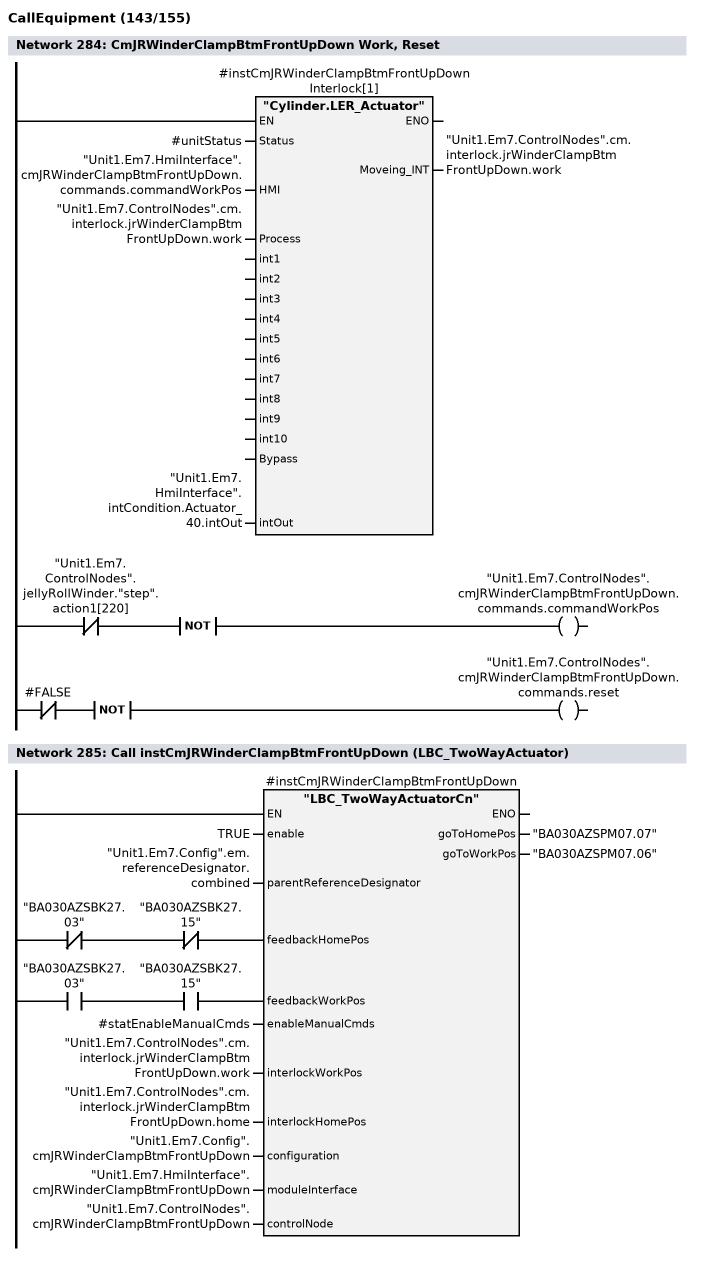
   RUNG wire#powerrail
      #instCmJRWinderClampBtmFrontUpDownInterlock[1](Status := #unitStatus, HMI := "Unit1.Em7.HmiInterface".cmJRWinderClampBtmFrontUpDown.commands.commandWorkPos, Process := "Unit1.Em7.ControlNodes".cm.interlock.jrWinderClampBtmFrontUpDown.work, int1 :=, int2 :=, int3 :=, int4 :=, int5 :=, int6 :=, int7 :=, int8 :=, int9 :=, int10 :=, Bypass :=, intOut := "Unit1.Em7.HmiInterface".intCondition.Actuator_40.intOut, Moveing_INT => "Unit1.Em7.ControlNodes".cm.interlock.jrWinderClampBtmFrontUpDown.work)
   END_RUNG
   RUNG wire#powerrail
      I_Contact( "Unit1.Em7.ControlNodes".jellyRollWinder."step".action1[220] )
      Not()
      Coil( "Unit1.Em7.ControlNodes".cmJRWinderClampBtmFrontUpDown.commands.commandWorkPos )
   END_RUNG
   RUNG wire#powerrail
      I_Contact( #FALSE )
      Not()
      Coil( "Unit1.Em7.ControlNodes".cmJRWinderClampBtmFrontUpDown.commands.reset )
   END_RUNG
   // the same network as SCL:
   #instCmJRWinderClampBtmFrontUpDownInterlock[1](Status := #unitStatus,   // "Cylinder.LER_Actuator"
                           HMI := "Unit1.Em7.HmiInterface".cmJRWinderClampBtmFrontUpDown.commands.commandWorkPos,
                           Process := "Unit1.Em7.ControlNodes".cm.interlock.jrWinderClampBtmFrontUpDown.work,
                           intOut := "Unit1.Em7.HmiInterface".intCondition.Actuator_40.intOut,
                           Moveing_INT => "Unit1.Em7.ControlNodes".cm.interlock.jrWinderClampBtmFrontUpDown.work);
   "Unit1.Em7.ControlNodes".cmJRWinderClampBtmFrontUpDown.commands.commandWorkPos := NOT (NOT "Unit1.Em7.ControlNodes".jellyRollWinder."step".action1[220]);
   "Unit1.Em7.ControlNodes".cmJRWinderClampBtmFrontUpDown.commands.reset := NOT (NOT #FALSE);
END_REGION

REGION Network 285: Call instCmJRWinderClampBtmFrontUpDown (LBC_TwoWayActuator)
   RUNG wire#powerrail
      #instCmJRWinderClampBtmFrontUpDown(feedbackHomePos := wire#w1, feedbackWorkPos := wire#w2, enable := TRUE, parentReferenceDesignator := "Unit1.Em7.Config".em.referenceDesignator.combined, enableManualCmds := #statEnableManualCmds, interlockWorkPos := "Unit1.Em7.ControlNodes".cm.interlock.jrWinderClampBtmFrontUpDown.work, interlockHomePos := "Unit1.Em7.ControlNodes".cm.interlock.jrWinderClampBtmFrontUpDown.home, configuration := "Unit1.Em7.Config".cmJRWinderClampBtmFrontUpDown, moduleInterface := "Unit1.Em7.HmiInterface".cmJRWinderClampBtmFrontUpDown, controlNode := "Unit1.Em7.ControlNodes".cmJRWinderClampBtmFrontUpDown, goToHomePos => "BA030AZSPM07.07", goToWorkPos => "BA030AZSPM07.06")
   END_RUNG
   RUNG wire#powerrail
      I_Contact( "BA030AZSBK27.03" )
      I_Contact( "BA030AZSBK27.15" )
   END_RUNG wire#w1
   RUNG wire#powerrail
      Contact( "BA030AZSBK27.03" )
      Contact( "BA030AZSBK27.15" )
   END_RUNG wire#w2
   // the same network as SCL:
   #instCmJRWinderClampBtmFrontUpDown(enable := TRUE,   // "LBC_TwoWayActuatorCn"
                           parentReferenceDesignator := "Unit1.Em7.Config".em.referenceDesignator.combined,
                           feedbackHomePos := NOT "BA030AZSBK27.03" AND NOT "BA030AZSBK27.15",
                           feedbackWorkPos := "BA030AZSBK27.03" AND "BA030AZSBK27.15",
                           enableManualCmds := #statEnableManualCmds,
                           interlockWorkPos := "Unit1.Em7.ControlNodes".cm.interlock.jrWinderClampBtmFrontUpDown.work,
                           interlockHomePos := "Unit1.Em7.ControlNodes".cm.interlock.jrWinderClampBtmFrontUpDown.home,
                           configuration := "Unit1.Em7.Config".cmJRWinderClampBtmFrontUpDown,
                           moduleInterface := "Unit1.Em7.HmiInterface".cmJRWinderClampBtmFrontUpDown,
                           controlNode := "Unit1.Em7.ControlNodes".cmJRWinderClampBtmFrontUpDown,
                           goToHomePos => "BA030AZSPM07.07",
                           goToWorkPos => "BA030AZSPM07.06");
END_REGION

REGION Network 287: CmPusherRollerFwdBwd Home
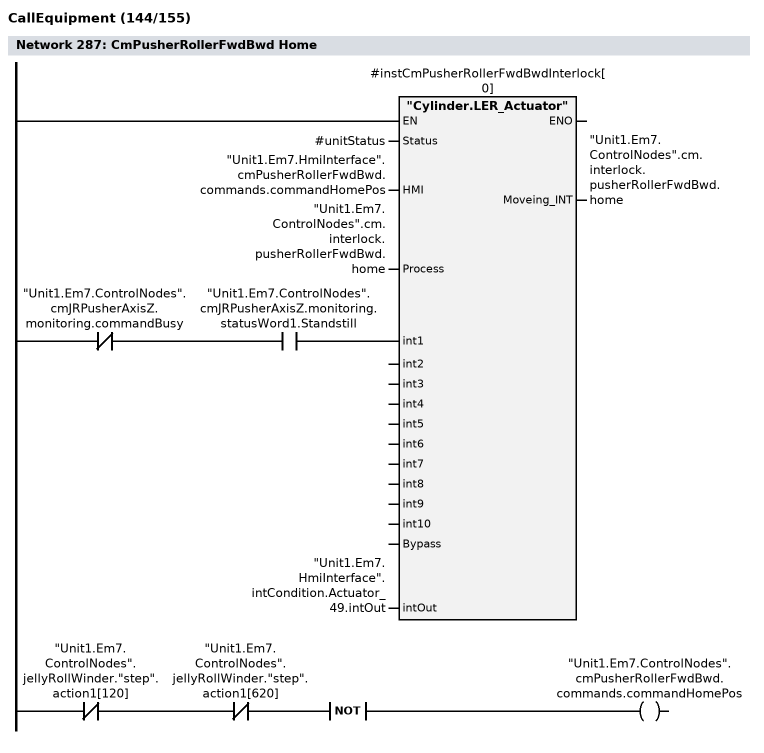
   RUNG wire#powerrail
      #instCmPusherRollerFwdBwdInterlock[0](int1 := wire#w1, Status := #unitStatus, HMI := "Unit1.Em7.HmiInterface".cmPusherRollerFwdBwd.commands.commandHomePos, Process := "Unit1.Em7.ControlNodes".cm.interlock.pusherRollerFwdBwd.home, int2 :=, int3 :=, int4 :=, int5 :=, int6 :=, int7 :=, int8 :=, int9 :=, int10 :=, Bypass :=, intOut := "Unit1.Em7.HmiInterface".intCondition.Actuator_49.intOut, Moveing_INT => "Unit1.Em7.ControlNodes".cm.interlock.pusherRollerFwdBwd.home)
   END_RUNG
   RUNG wire#powerrail
      I_Contact( "Unit1.Em7.ControlNodes".cmJRPusherAxisZ.monitoring.commandBusy )
      Contact( "Unit1.Em7.ControlNodes".cmJRPusherAxisZ.monitoring.statusWord1.Standstill )
   END_RUNG wire#w1
   RUNG wire#powerrail
      I_Contact( "Unit1.Em7.ControlNodes".jellyRollWinder."step".action1[120] )
      I_Contact( "Unit1.Em7.ControlNodes".jellyRollWinder."step".action1[620] )
      Not()
      Coil( "Unit1.Em7.ControlNodes".cmPusherRollerFwdBwd.commands.commandHomePos )
   END_RUNG
   // the same network as SCL:
   #instCmPusherRollerFwdBwdInterlock[0](Status := #unitStatus,   // "Cylinder.LER_Actuator"
                           HMI := "Unit1.Em7.HmiInterface".cmPusherRollerFwdBwd.commands.commandHomePos,
                           Process := "Unit1.Em7.ControlNodes".cm.interlock.pusherRollerFwdBwd.home,
                           int1 := NOT "Unit1.Em7.ControlNodes".cmJRPusherAxisZ.monitoring.commandBusy AND "Unit1.Em7.ControlNodes".cmJRPusherAxisZ.monitoring.statusWord1.Standstill,
                           intOut := "Unit1.Em7.HmiInterface".intCondition.Actuator_49.intOut,
                           Moveing_INT => "Unit1.Em7.ControlNodes".cm.interlock.pusherRollerFwdBwd.home);
   "Unit1.Em7.ControlNodes".cmPusherRollerFwdBwd.commands.commandHomePos := NOT (NOT "Unit1.Em7.ControlNodes".jellyRollWinder."step".action1[120] AND NOT "Unit1.Em7.ControlNodes".jellyRollWinder."step".action1[620]);
END_REGION

REGION Network 288: CmPusherRollerFwdBwd Work
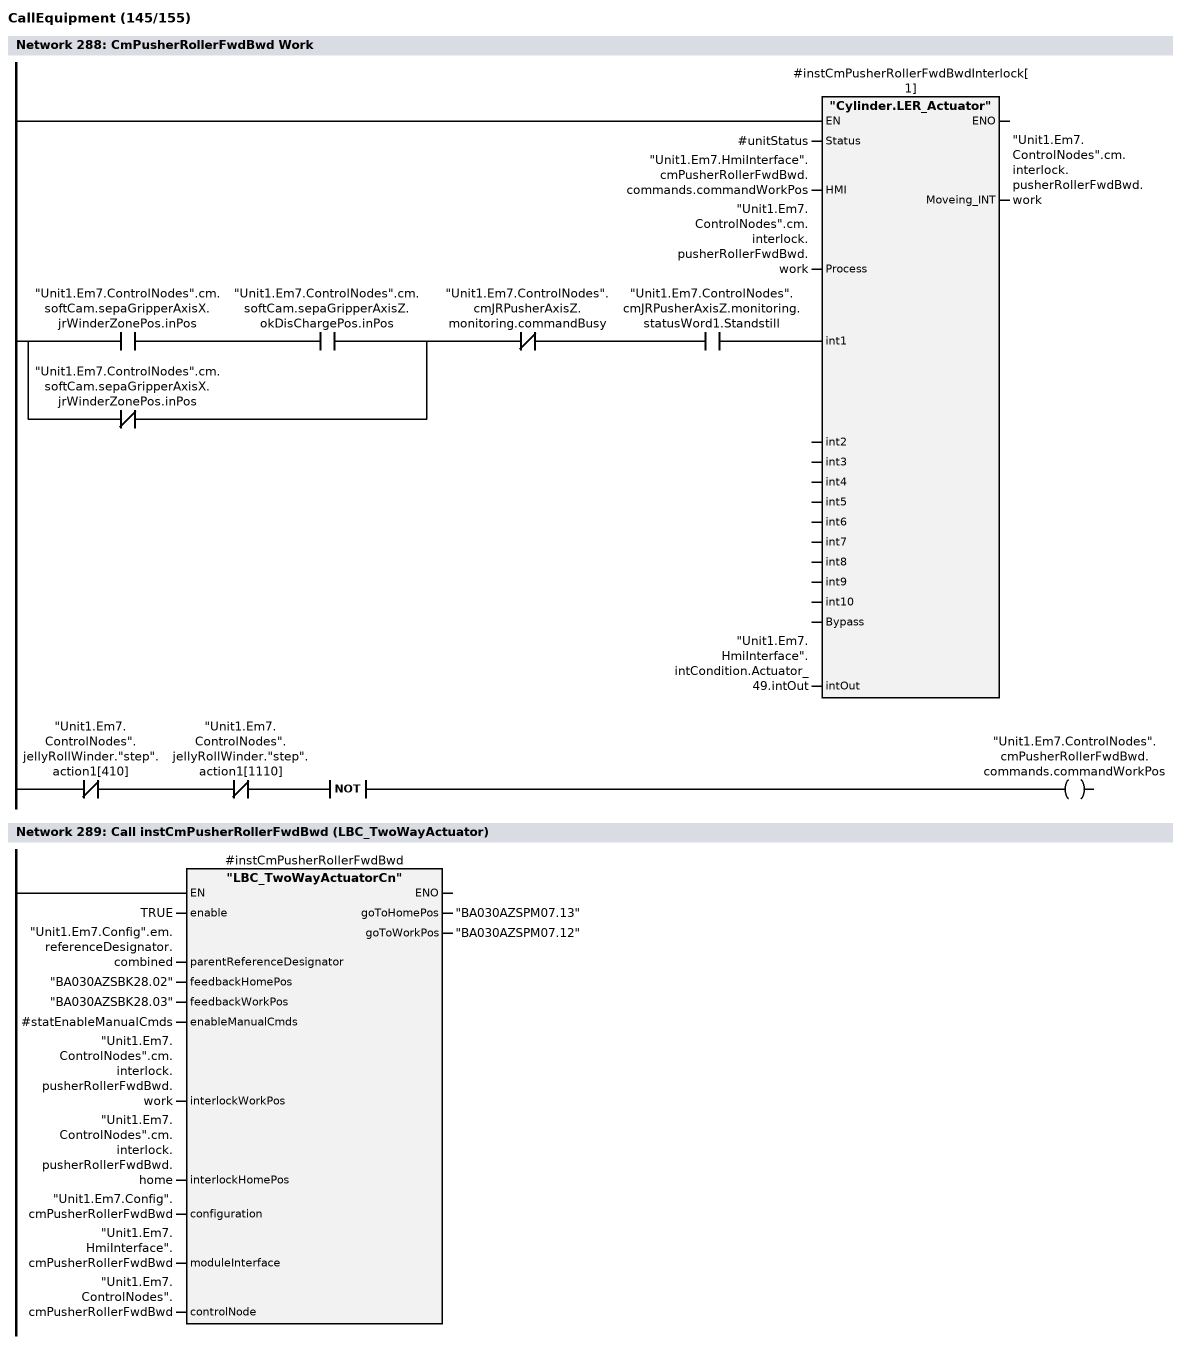
   RUNG wire#powerrail
      #instCmPusherRollerFwdBwdInterlock[1](int1 := wire#w2, Status := #unitStatus, HMI := "Unit1.Em7.HmiInterface".cmPusherRollerFwdBwd.commands.commandWorkPos, Process := "Unit1.Em7.ControlNodes".cm.interlock.pusherRollerFwdBwd.work, int2 :=, int3 :=, int4 :=, int5 :=, int6 :=, int7 :=, int8 :=, int9 :=, int10 :=, Bypass :=, intOut := "Unit1.Em7.HmiInterface".intCondition.Actuator_49.intOut, Moveing_INT => "Unit1.Em7.ControlNodes".cm.interlock.pusherRollerFwdBwd.work)
   END_RUNG
   RUNG wire#powerrail
      Contact( "Unit1.Em7.ControlNodes".cm.softCam.sepaGripperAxisX.jrWinderZonePos.inPos )
      Contact( "Unit1.Em7.ControlNodes".cm.softCam.sepaGripperAxisZ.okDisChargePos.inPos )
      wire#w1
      I_Contact( "Unit1.Em7.ControlNodes".cmJRPusherAxisZ.monitoring.commandBusy )
      Contact( "Unit1.Em7.ControlNodes".cmJRPusherAxisZ.monitoring.statusWord1.Standstill )
   END_RUNG wire#w2
   RUNG wire#powerrail
      I_Contact( "Unit1.Em7.ControlNodes".cm.softCam.sepaGripperAxisX.jrWinderZonePos.inPos )
   END_RUNG wire#w1
   RUNG wire#powerrail
      I_Contact( "Unit1.Em7.ControlNodes".jellyRollWinder."step".action1[410] )
      I_Contact( "Unit1.Em7.ControlNodes".jellyRollWinder."step".action1[1110] )
      Not()
      Coil( "Unit1.Em7.ControlNodes".cmPusherRollerFwdBwd.commands.commandWorkPos )
   END_RUNG
   // the same network as SCL:
   #instCmPusherRollerFwdBwdInterlock[1](Status := #unitStatus,   // "Cylinder.LER_Actuator"
                           HMI := "Unit1.Em7.HmiInterface".cmPusherRollerFwdBwd.commands.commandWorkPos,
                           Process := "Unit1.Em7.ControlNodes".cm.interlock.pusherRollerFwdBwd.work,
                           int1 := (("Unit1.Em7.ControlNodes".cm.softCam.sepaGripperAxisX.jrWinderZonePos.inPos AND "Unit1.Em7.ControlNodes".cm.softCam.sepaGripperAxisZ.okDisChargePos.inPos) OR NOT "Unit1.Em7.ControlNodes".cm.softCam.sepaGripperAxisX.jrWinderZonePos.inPos) AND NOT "Unit1.Em7.ControlNodes".cmJRPusherAxisZ.monitoring.commandBusy AND "Unit1.Em7.ControlNodes".cmJRPusherAxisZ.monitoring.statusWord1.Standstill,
                           intOut := "Unit1.Em7.HmiInterface".intCondition.Actuator_49.intOut,
                           Moveing_INT => "Unit1.Em7.ControlNodes".cm.interlock.pusherRollerFwdBwd.work);
   "Unit1.Em7.ControlNodes".cmPusherRollerFwdBwd.commands.commandWorkPos := NOT (NOT "Unit1.Em7.ControlNodes".jellyRollWinder."step".action1[410] AND NOT "Unit1.Em7.ControlNodes".jellyRollWinder."step".action1[1110]);
END_REGION

REGION Network 289: Call instCmPusherRollerFwdBwd (LBC_TwoWayActuator)
   RUNG wire#powerrail
      #instCmPusherRollerFwdBwd(enable := TRUE, parentReferenceDesignator := "Unit1.Em7.Config".em.referenceDesignator.combined, feedbackHomePos := "BA030AZSBK28.02", feedbackWorkPos := "BA030AZSBK28.03", enableManualCmds := #statEnableManualCmds, interlockWorkPos := "Unit1.Em7.ControlNodes".cm.interlock.pusherRollerFwdBwd.work, interlockHomePos := "Unit1.Em7.ControlNodes".cm.interlock.pusherRollerFwdBwd.home, configuration := "Unit1.Em7.Config".cmPusherRollerFwdBwd, moduleInterface := "Unit1.Em7.HmiInterface".cmPusherRollerFwdBwd, controlNode := "Unit1.Em7.ControlNodes".cmPusherRollerFwdBwd, goToHomePos => "BA030AZSPM07.13", goToWorkPos => "BA030AZSPM07.12")
   END_RUNG
   // the same network as SCL:
   #instCmPusherRollerFwdBwd(enable := TRUE,   // "LBC_TwoWayActuatorCn"
                           parentReferenceDesignator := "Unit1.Em7.Config".em.referenceDesignator.combined,
                           feedbackHomePos := "BA030AZSBK28.02",
                           feedbackWorkPos := "BA030AZSBK28.03",
                           enableManualCmds := #statEnableManualCmds,
                           interlockWorkPos := "Unit1.Em7.ControlNodes".cm.interlock.pusherRollerFwdBwd.work,
                           interlockHomePos := "Unit1.Em7.ControlNodes".cm.interlock.pusherRollerFwdBwd.home,
                           configuration := "Unit1.Em7.Config".cmPusherRollerFwdBwd,
                           moduleInterface := "Unit1.Em7.HmiInterface".cmPusherRollerFwdBwd,
                           controlNode := "Unit1.Em7.ControlNodes".cmPusherRollerFwdBwd,
                           goToHomePos => "BA030AZSPM07.13",
                           goToWorkPos => "BA030AZSPM07.12");
END_REGION

REGION Network 291: ********** Feedback to Unit **********
END_REGION

REGION Network 292: Determine StateComplete (SC) in Mode Production
   // Conditions for the Equipment Modules "stateComplete" feedback to the unit. This feedback is given when the task in for the respective state is complete.
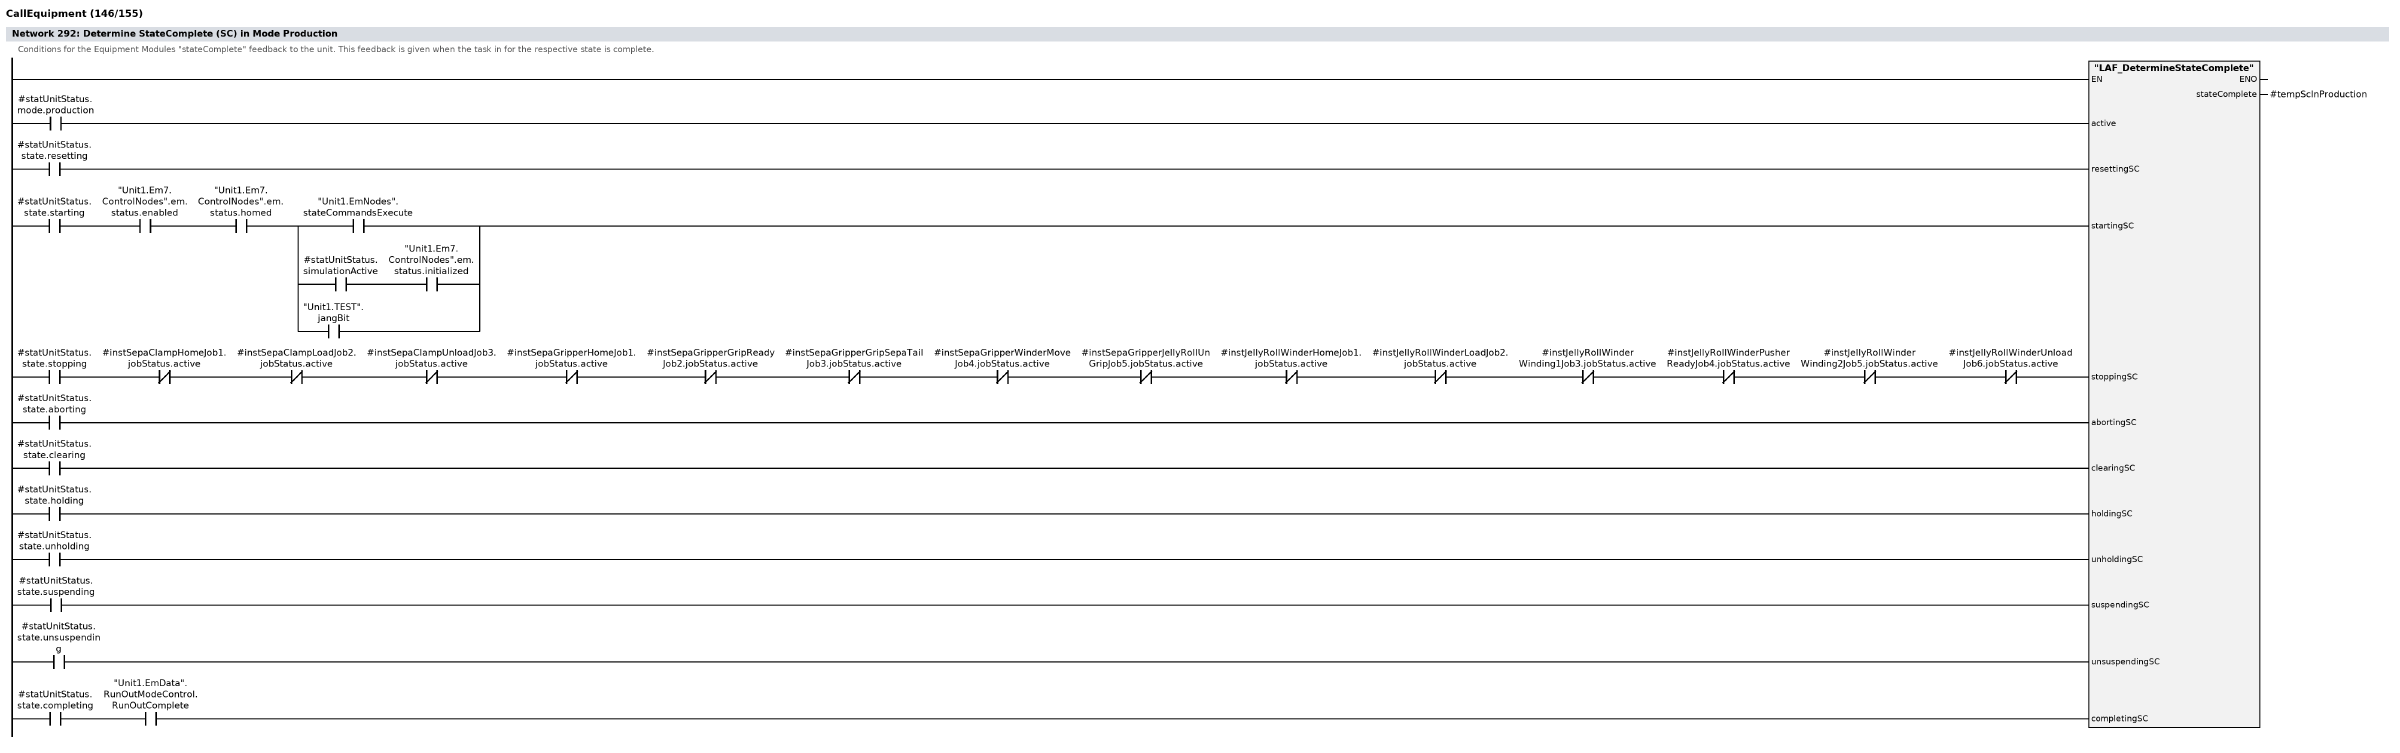
   RUNG wire#powerrail
      "LAF_DetermineStateComplete"(active := wire#w1, resettingSC := wire#w2, startingSC := wire#w4, stoppingSC := wire#w5, abortingSC := wire#w6, clearingSC := wire#w7, holdingSC := wire#w8, unholdingSC := wire#w9, suspendingSC := wire#w10, unsuspendingSC := wire#w11, completingSC := wire#w12, stateComplete => #tempScInProduction)
   END_RUNG
   RUNG wire#powerrail
      Contact( #statUnitStatus.mode.production )
   END_RUNG wire#w1
   RUNG wire#powerrail
      Contact( #statUnitStatus.state.resetting )
   END_RUNG wire#w2
   RUNG wire#powerrail
      Contact( #statUnitStatus.state.starting )
      Contact( "Unit1.Em7.ControlNodes".em.status.enabled )
      Contact( "Unit1.Em7.ControlNodes".em.status.homed )
      wire#w3
      Contact( "Unit1.EmNodes".stateCommandsExecute )
   END_RUNG wire#w4
   RUNG wire#w3
      Contact( #statUnitStatus.simulationActive )
      Contact( "Unit1.Em7.ControlNodes".em.status.initialized )
   END_RUNG wire#w4
   RUNG wire#w3
      Contact( "Unit1.TEST".jangBit )
   END_RUNG wire#w4
   RUNG wire#powerrail
      Contact( #statUnitStatus.state.stopping )
      I_Contact( #instSepaClampHomeJob1.jobStatus.active )
      I_Contact( #instSepaClampLoadJob2.jobStatus.active )
      I_Contact( #instSepaClampUnloadJob3.jobStatus.active )
      I_Contact( #instSepaGripperHomeJob1.jobStatus.active )
      I_Contact( #instSepaGripperGripReadyJob2.jobStatus.active )
      I_Contact( #instSepaGripperGripSepaTailJob3.jobStatus.active )
      I_Contact( #instSepaGripperWinderMoveJob4.jobStatus.active )
      I_Contact( #instSepaGripperJellyRollUnGripJob5.jobStatus.active )
      I_Contact( #instJellyRollWinderHomeJob1.jobStatus.active )
      I_Contact( #instJellyRollWinderLoadJob2.jobStatus.active )
      I_Contact( #instJellyRollWinderWinding1Job3.jobStatus.active )
      I_Contact( #instJellyRollWinderPusherReadyJob4.jobStatus.active )
      I_Contact( #instJellyRollWinderWinding2Job5.jobStatus.active )
      I_Contact( #instJellyRollWinderUnloadJob6.jobStatus.active )
   END_RUNG wire#w5
   RUNG wire#powerrail
      Contact( #statUnitStatus.state.aborting )
   END_RUNG wire#w6
   RUNG wire#powerrail
      Contact( #statUnitStatus.state.clearing )
   END_RUNG wire#w7
   RUNG wire#powerrail
      Contact( #statUnitStatus.state.holding )
   END_RUNG wire#w8
   RUNG wire#powerrail
      Contact( #statUnitStatus.state.unholding )
   END_RUNG wire#w9
   RUNG wire#powerrail
      Contact( #statUnitStatus.state.suspending )
   END_RUNG wire#w10
   RUNG wire#powerrail
      Contact( #statUnitStatus.state.unsuspending )
   END_RUNG wire#w11
   RUNG wire#powerrail
      Contact( #statUnitStatus.state.completing )
      Contact( "Unit1.EmData".RunOutModeControl.RunOutComplete )
   END_RUNG wire#w12
   // the same network as SCL:
   "LAF_DetermineStateComplete"(active := #statUnitStatus.mode.production,
                           resettingSC := #statUnitStatus.state.resetting,
                           startingSC := #statUnitStatus.state.starting AND "Unit1.Em7.ControlNodes".em.status.enabled AND "Unit1.Em7.ControlNodes".em.status.homed AND ("Unit1.EmNodes".stateCommandsExecute OR (#statUnitStatus.simulationActive AND "Unit1.Em7.ControlNodes".em.status.initialized) OR "Unit1.TEST".jangBit),
                           stoppingSC := #statUnitStatus.state.stopping AND NOT #instSepaClampHomeJob1.jobStatus.active AND NOT #instSepaClampLoadJob2.jobStatus.active AND NOT #instSepaClampUnloadJob3.jobStatus.active AND NOT #instSepaGripperHomeJob1.jobStatus.active AND NOT #instSepaGripperGripReadyJob2.jobStatus.active AND NOT #instSepaGripperGripSepaTailJob3.jobStatus.active AND NOT #instSepaGripperWinderMoveJob4.jobStatus.active AND NOT #instSepaGripperJellyRollUnGripJob5.jobStatus.active AND NOT #instJellyRollWinderHomeJob1.jobStatus.active AND NOT #instJellyRollWinderLoadJob2.jobStatus.active AND NOT #instJellyRollWinderWinding1Job3.jobStatus.active AND NOT #instJellyRollWinderPusherReadyJob4.jobStatus.active AND NOT #instJellyRollWinderWinding2Job5.jobStatus.active AND NOT #instJellyRollWinderUnloadJob6.jobStatus.active,
                           abortingSC := #statUnitStatus.state.aborting,
                           clearingSC := #statUnitStatus.state.clearing,
                           holdingSC := #statUnitStatus.state.holding,
                           unholdingSC := #statUnitStatus.state.unholding,
                           suspendingSC := #statUnitStatus.state.suspending,
                           unsuspendingSC := #statUnitStatus.state.unsuspending,
                           completingSC := #statUnitStatus.state.completing AND "Unit1.EmData".RunOutModeControl.RunOutComplete,
                           stateComplete => #tempScInProduction);
END_REGION

REGION Network 293: Determine StateComplete (SC) in Mode Maintenance/Manual
   // Conditions for the Equipment Modules "stateComplete" feedback to the unit. This feedback is given when the task in for the respective state is complete.
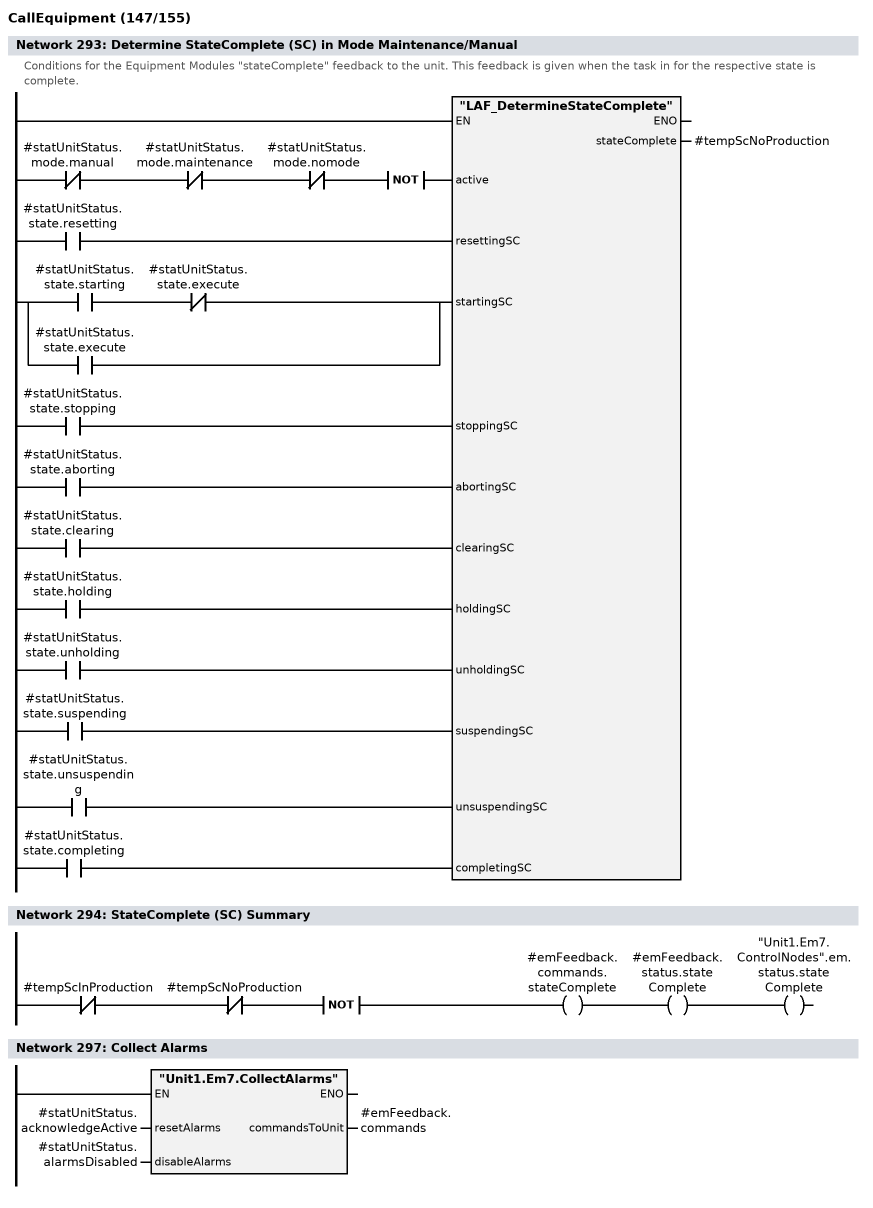
   RUNG wire#powerrail
      "LAF_DetermineStateComplete"(active := wire#w1, resettingSC := wire#w2, startingSC := wire#w3, stoppingSC := wire#w4, abortingSC := wire#w5, clearingSC := wire#w6, holdingSC := wire#w7, unholdingSC := wire#w8, suspendingSC := wire#w9, unsuspendingSC := wire#w10, completingSC := wire#w11, stateComplete => #tempScNoProduction)
   END_RUNG
   RUNG wire#powerrail
      I_Contact( #statUnitStatus.mode.manual )
      I_Contact( #statUnitStatus.mode.maintenance )
      I_Contact( #statUnitStatus.mode.nomode )
      Not()
   END_RUNG wire#w1
   RUNG wire#powerrail
      Contact( #statUnitStatus.state.resetting )
   END_RUNG wire#w2
   RUNG wire#powerrail
      Contact( #statUnitStatus.state.starting )
      I_Contact( #statUnitStatus.state.execute )
   END_RUNG wire#w3
   RUNG wire#powerrail
      Contact( #statUnitStatus.state.execute )
   END_RUNG wire#w3
   RUNG wire#powerrail
      Contact( #statUnitStatus.state.stopping )
   END_RUNG wire#w4
   RUNG wire#powerrail
      Contact( #statUnitStatus.state.aborting )
   END_RUNG wire#w5
   RUNG wire#powerrail
      Contact( #statUnitStatus.state.clearing )
   END_RUNG wire#w6
   RUNG wire#powerrail
      Contact( #statUnitStatus.state.holding )
   END_RUNG wire#w7
   RUNG wire#powerrail
      Contact( #statUnitStatus.state.unholding )
   END_RUNG wire#w8
   RUNG wire#powerrail
      Contact( #statUnitStatus.state.suspending )
   END_RUNG wire#w9
   RUNG wire#powerrail
      Contact( #statUnitStatus.state.unsuspending )
   END_RUNG wire#w10
   RUNG wire#powerrail
      Contact( #statUnitStatus.state.completing )
   END_RUNG wire#w11
   // the same network as SCL:
   "LAF_DetermineStateComplete"(active := NOT (NOT #statUnitStatus.mode.manual AND NOT #statUnitStatus.mode.maintenance AND NOT #statUnitStatus.mode.nomode),
                           resettingSC := #statUnitStatus.state.resetting,
                           startingSC := (#statUnitStatus.state.starting AND NOT #statUnitStatus.state.execute) OR #statUnitStatus.state.execute,
                           stoppingSC := #statUnitStatus.state.stopping,
                           abortingSC := #statUnitStatus.state.aborting,
                           clearingSC := #statUnitStatus.state.clearing,
                           holdingSC := #statUnitStatus.state.holding,
                           unholdingSC := #statUnitStatus.state.unholding,
                           suspendingSC := #statUnitStatus.state.suspending,
                           unsuspendingSC := #statUnitStatus.state.unsuspending,
                           completingSC := #statUnitStatus.state.completing,
                           stateComplete => #tempScNoProduction);
END_REGION

REGION Network 294: StateComplete (SC) Summary
   RUNG wire#powerrail
      I_Contact( #tempScInProduction )
      I_Contact( #tempScNoProduction )
      Not()
      Coil( #emFeedback.commands.stateComplete )
      Coil( #emFeedback.status.stateComplete )
      Coil( "Unit1.Em7.ControlNodes".em.status.stateComplete )
   END_RUNG
   // the same network as SCL:
   #emFeedback.commands.stateComplete := NOT (NOT #tempScInProduction AND NOT #tempScNoProduction);
   #emFeedback.status.stateComplete := #emFeedback.commands.stateComplete;
   "Unit1.Em7.ControlNodes".em.status.stateComplete := #emFeedback.commands.stateComplete;
END_REGION

REGION Network 296: ********** Alarms **********
END_REGION

REGION Network 297: Collect Alarms
   RUNG wire#powerrail
      "Unit1.Em7.CollectAlarms"(resetAlarms := #statUnitStatus.acknowledgeActive, disableAlarms := #statUnitStatus.alarmsDisabled, commandsToUnit => #emFeedback.commands)
   END_RUNG
   // the same network as SCL:
   "Unit1.Em7.CollectAlarms"(resetAlarms := #statUnitStatus.acknowledgeActive,
                           disableAlarms := #statUnitStatus.alarmsDisabled,
                           commandsToUnit => #emFeedback.commands);
END_REGION

REGION Network 298: Manage Alarms
   // Derive commands from the ProDiag supervision. The ProDiag supervisions contain categories which define the reaction of these supervisions (e.g. abort, stop, hold). These are handed over as commands to the unit level.
   // Alternatively, if no ProDiag should be used, you can use the LAF_ManageBitAlarms to realize bit alarm handling. This block can be found in LAF in folder 70_AlarmHandling.
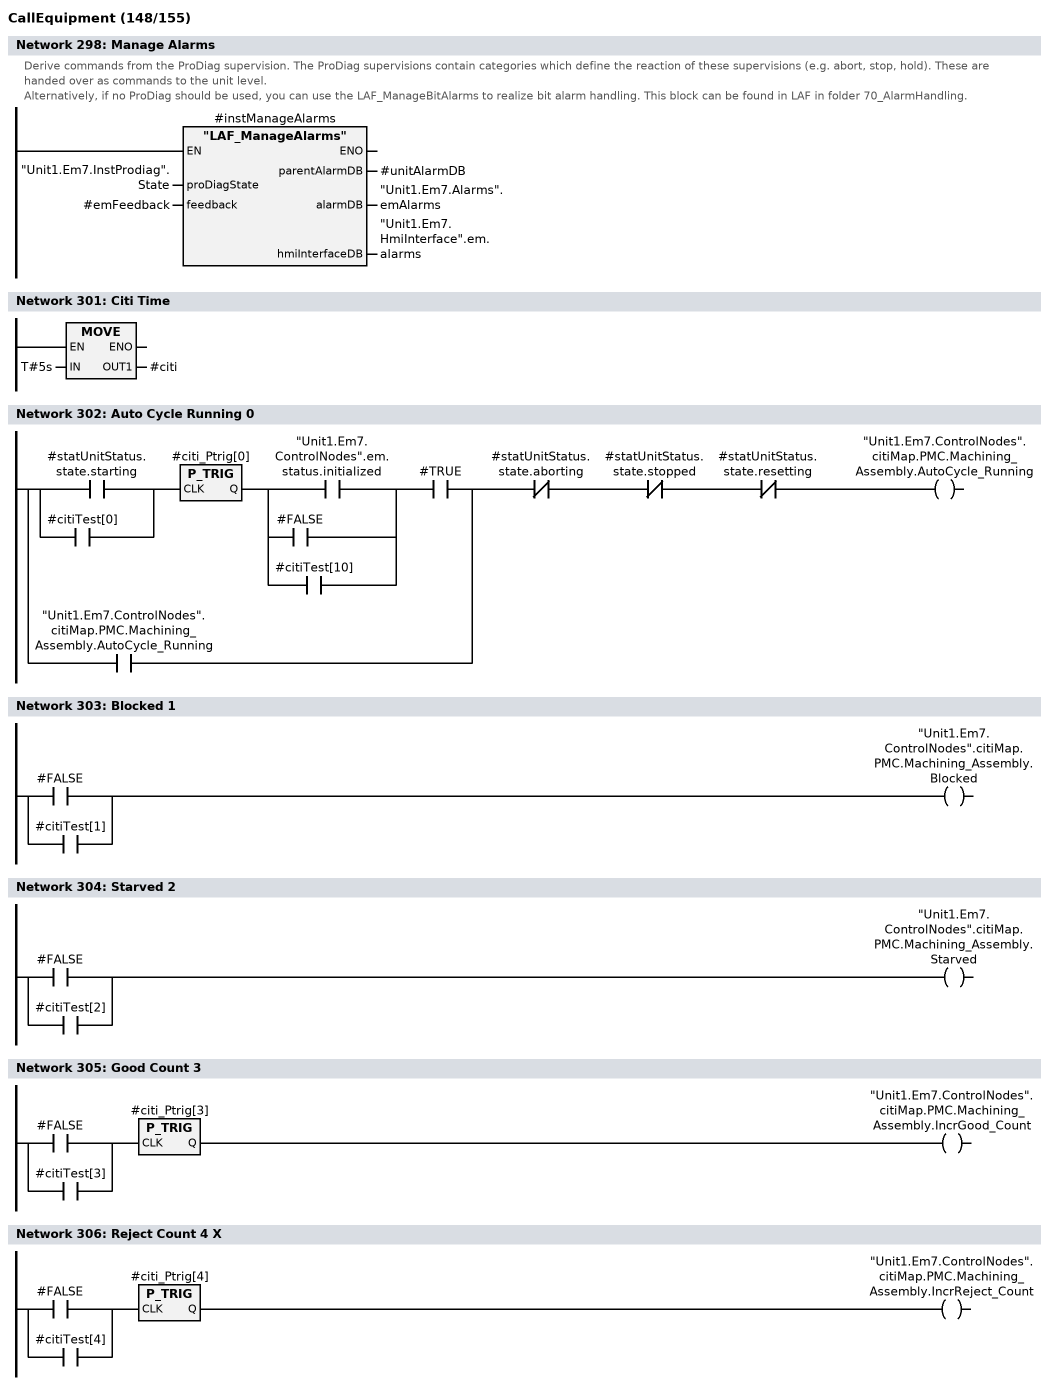
   RUNG wire#powerrail
      #instManageAlarms(proDiagState := "Unit1.Em7.InstProdiag".State, feedback := #emFeedback, parentAlarmDB => #unitAlarmDB, alarmDB => "Unit1.Em7.Alarms".emAlarms, hmiInterfaceDB => "Unit1.Em7.HmiInterface".em.alarms)
   END_RUNG
   // the same network as SCL:
   #instManageAlarms(proDiagState := "Unit1.Em7.InstProdiag".State,   // "LAF_ManageAlarms"
                     feedback := #emFeedback,
                     parentAlarmDB => #unitAlarmDB,
                     alarmDB => "Unit1.Em7.Alarms".emAlarms,
                     hmiInterfaceDB => "Unit1.Em7.HmiInterface".em.alarms);
END_REGION

REGION Network 300: ******************** CITI ********************
END_REGION

REGION Network 301: Citi Time
   RUNG wire#powerrail
      Move(in := T#5s, out1 => #citi)
   END_RUNG
   // the same network as SCL:
   #citi := T#5s;
END_REGION

REGION Network 302: Auto Cycle Running 0
   RUNG wire#powerrail
      Contact( #statUnitStatus.state.starting )
      wire#w1
      P_Trig( #citi_Ptrig[0] )
      wire#w2
      Contact( "Unit1.Em7.ControlNodes".em.status.initialized )
      wire#w3
      Contact( #TRUE )
      wire#w4
      I_Contact( #statUnitStatus.state.aborting )
      I_Contact( #statUnitStatus.state.stopped )
      I_Contact( #statUnitStatus.state.resetting )
      Coil( "Unit1.Em7.ControlNodes".citiMap.PMC.Machining_Assembly.AutoCycle_Running )
   END_RUNG
   RUNG wire#powerrail
      Contact( #citiTest[0] )
   END_RUNG wire#w1
   RUNG wire#w2
      Contact( #FALSE )
   END_RUNG wire#w3
   RUNG wire#w2
      Contact( #citiTest[10] )
   END_RUNG wire#w3
   RUNG wire#powerrail
      Contact( "Unit1.Em7.ControlNodes".citiMap.PMC.Machining_Assembly.AutoCycle_Running )
   END_RUNG wire#w4
   // the same network as SCL:
   #_w1 := #statUnitStatus.state.starting OR #citiTest[0];
   #_w2 := #_w1 AND NOT #citi_Ptrig[0];   // rising edge
   #citi_Ptrig[0] := #_w1;
   "Unit1.Em7.ControlNodes".citiMap.PMC.Machining_Assembly.AutoCycle_Running := ((#_w2 AND ("Unit1.Em7.ControlNodes".em.status.initialized OR #FALSE OR #citiTest[10]) AND #TRUE) OR "Unit1.Em7.ControlNodes".citiMap.PMC.Machining_Assembly.AutoCycle_Running) AND NOT #statUnitStatus.state.aborting AND NOT #statUnitStatus.state.stopped AND NOT #statUnitStatus.state.resetting;
END_REGION

REGION Network 303: Blocked 1
   RUNG wire#powerrail
      Contact( #FALSE )
      wire#w1
      Coil( "Unit1.Em7.ControlNodes".citiMap.PMC.Machining_Assembly.Blocked )
   END_RUNG
   RUNG wire#powerrail
      Contact( #citiTest[1] )
   END_RUNG wire#w1
   // the same network as SCL:
   "Unit1.Em7.ControlNodes".citiMap.PMC.Machining_Assembly.Blocked := #FALSE OR #citiTest[1];
END_REGION

REGION Network 304: Starved 2
   RUNG wire#powerrail
      Contact( #FALSE )
      wire#w1
      Coil( "Unit1.Em7.ControlNodes".citiMap.PMC.Machining_Assembly.Starved )
   END_RUNG
   RUNG wire#powerrail
      Contact( #citiTest[2] )
   END_RUNG wire#w1
   // the same network as SCL:
   "Unit1.Em7.ControlNodes".citiMap.PMC.Machining_Assembly.Starved := #FALSE OR #citiTest[2];
END_REGION

REGION Network 305: Good Count 3
   RUNG wire#powerrail
      Contact( #FALSE )
      wire#w1
      P_Trig( #citi_Ptrig[3] )
      Coil( "Unit1.Em7.ControlNodes".citiMap.PMC.Machining_Assembly.IncrGood_Count )
   END_RUNG
   RUNG wire#powerrail
      Contact( #citiTest[3] )
   END_RUNG wire#w1
   // the same network as SCL:
   #_w1 := #FALSE OR #citiTest[3];
   #_w2 := #_w1 AND NOT #citi_Ptrig[3];   // rising edge
   #citi_Ptrig[3] := #_w1;
   "Unit1.Em7.ControlNodes".citiMap.PMC.Machining_Assembly.IncrGood_Count := #_w2;
END_REGION

REGION Network 306: Reject Count 4 X
   RUNG wire#powerrail
      Contact( #FALSE )
      wire#w1
      P_Trig( #citi_Ptrig[4] )
      Coil( "Unit1.Em7.ControlNodes".citiMap.PMC.Machining_Assembly.IncrReject_Count )
   END_RUNG
   RUNG wire#powerrail
      Contact( #citiTest[4] )
   END_RUNG wire#w1
   // the same network as SCL:
   #_w1 := #FALSE OR #citiTest[4];
   #_w2 := #_w1 AND NOT #citi_Ptrig[4];   // rising edge
   #citi_Ptrig[4] := #_w1;
   "Unit1.Em7.ControlNodes".citiMap.PMC.Machining_Assembly.IncrReject_Count := #_w2;
END_REGION

REGION Network 307: Cycle End Trigger 5
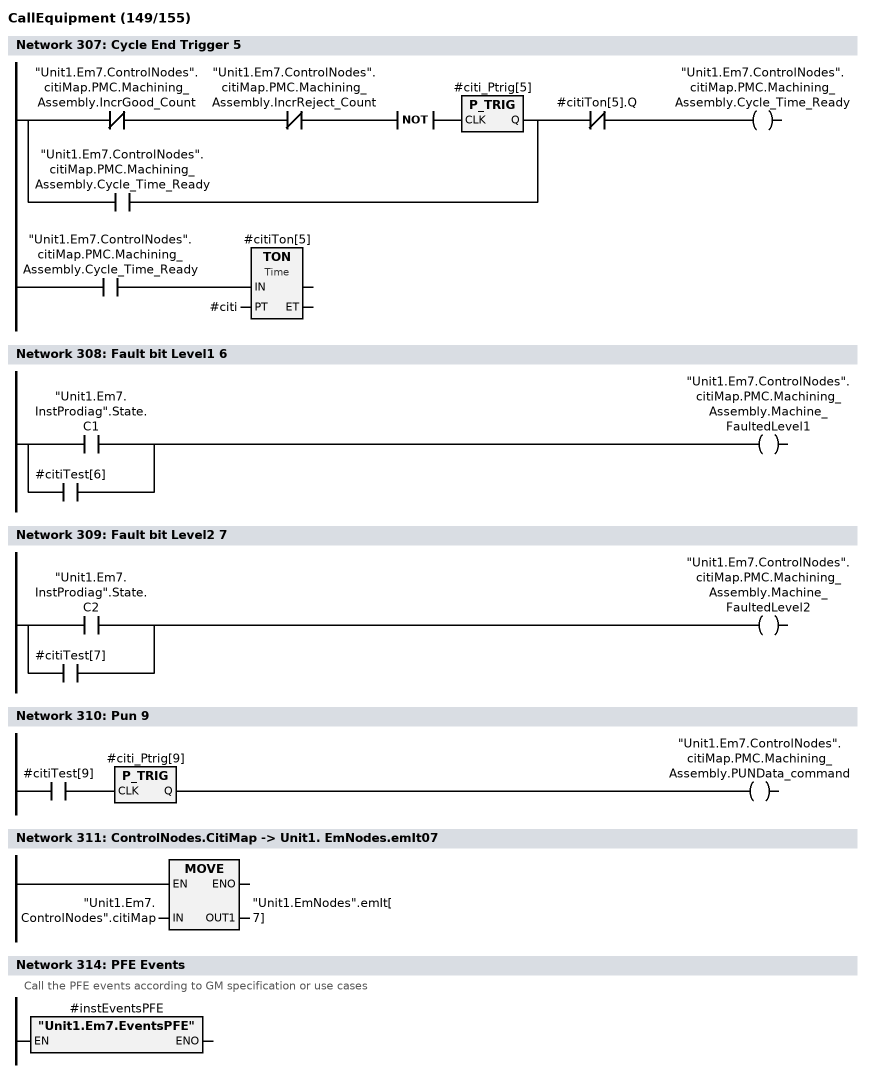
   RUNG wire#powerrail
      I_Contact( "Unit1.Em7.ControlNodes".citiMap.PMC.Machining_Assembly.IncrGood_Count )
      I_Contact( "Unit1.Em7.ControlNodes".citiMap.PMC.Machining_Assembly.IncrReject_Count )
      Not()
      P_Trig( #citi_Ptrig[5] )
      wire#w1
      I_Contact( #citiTon[5].Q )
      Coil( "Unit1.Em7.ControlNodes".citiMap.PMC.Machining_Assembly.Cycle_Time_Ready )
   END_RUNG
   RUNG wire#powerrail
      Contact( "Unit1.Em7.ControlNodes".citiMap.PMC.Machining_Assembly.Cycle_Time_Ready )
   END_RUNG wire#w1
   RUNG wire#powerrail
      Contact( "Unit1.Em7.ControlNodes".citiMap.PMC.Machining_Assembly.Cycle_Time_Ready )
      { S7_Templates := "time_type := Time" } #citiTon[5].TON(pt := #citi, et =>)
   END_RUNG
   // the same network as SCL:
   #_w1 := NOT (NOT "Unit1.Em7.ControlNodes".citiMap.PMC.Machining_Assembly.IncrGood_Count AND NOT "Unit1.Em7.ControlNodes".citiMap.PMC.Machining_Assembly.IncrReject_Count);
   #_w2 := #_w1 AND NOT #citi_Ptrig[5];   // rising edge
   #citi_Ptrig[5] := #_w1;
   "Unit1.Em7.ControlNodes".citiMap.PMC.Machining_Assembly.Cycle_Time_Ready := (#_w2 OR "Unit1.Em7.ControlNodes".citiMap.PMC.Machining_Assembly.Cycle_Time_Ready) AND NOT #citiTon[5].Q;
   #citiTon[5].TON(IN := "Unit1.Em7.ControlNodes".citiMap.PMC.Machining_Assembly.Cycle_Time_Ready, PT := #citi);
END_REGION

REGION Network 308: Fault bit Level1 6
   RUNG wire#powerrail
      Contact( "Unit1.Em7.InstProdiag".State.C1 )
      wire#w1
      Coil( "Unit1.Em7.ControlNodes".citiMap.PMC.Machining_Assembly.Machine_FaultedLevel1 )
   END_RUNG
   RUNG wire#powerrail
      Contact( #citiTest[6] )
   END_RUNG wire#w1
   // the same network as SCL:
   "Unit1.Em7.ControlNodes".citiMap.PMC.Machining_Assembly.Machine_FaultedLevel1 := "Unit1.Em7.InstProdiag".State.C1 OR #citiTest[6];
END_REGION

REGION Network 309: Fault bit Level2 7
   RUNG wire#powerrail
      Contact( "Unit1.Em7.InstProdiag".State.C2 )
      wire#w1
      Coil( "Unit1.Em7.ControlNodes".citiMap.PMC.Machining_Assembly.Machine_FaultedLevel2 )
   END_RUNG
   RUNG wire#powerrail
      Contact( #citiTest[7] )
   END_RUNG wire#w1
   // the same network as SCL:
   "Unit1.Em7.ControlNodes".citiMap.PMC.Machining_Assembly.Machine_FaultedLevel2 := "Unit1.Em7.InstProdiag".State.C2 OR #citiTest[7];
END_REGION

REGION Network 310: Pun 9
   RUNG wire#powerrail
      Contact( #citiTest[9] )
      P_Trig( #citi_Ptrig[9] )
      Coil( "Unit1.Em7.ControlNodes".citiMap.PMC.Machining_Assembly.PUNData_command )
   END_RUNG
   // the same network as SCL:
   #_w1 := #citiTest[9] AND NOT #citi_Ptrig[9];   // rising edge
   #citi_Ptrig[9] := #citiTest[9];
   "Unit1.Em7.ControlNodes".citiMap.PMC.Machining_Assembly.PUNData_command := #_w1;
END_REGION

REGION Network 311: ControlNodes.CitiMap -> Unit1. EmNodes.emIt07
   RUNG wire#powerrail
      Move(in := "Unit1.Em7.ControlNodes".citiMap, out1 => "Unit1.EmNodes".emIt[7])
   END_RUNG
   // the same network as SCL:
   "Unit1.EmNodes".emIt[7] := "Unit1.Em7.ControlNodes".citiMap;
END_REGION

REGION Network 313: ********** PFE Events **********
END_REGION

REGION Network 314: PFE Events
   // Call the PFE events according to GM specification or use cases
   RUNG wire#powerrail
      #instEventsPFE()
   END_RUNG
   // the same network as SCL:
   #instEventsPFE();   // "Unit1.Em7.EventsPFE"
END_REGION

REGION Network 316: ******************** Unit Output ********************
END_REGION

REGION Network 317: Em7 Relations Softcam
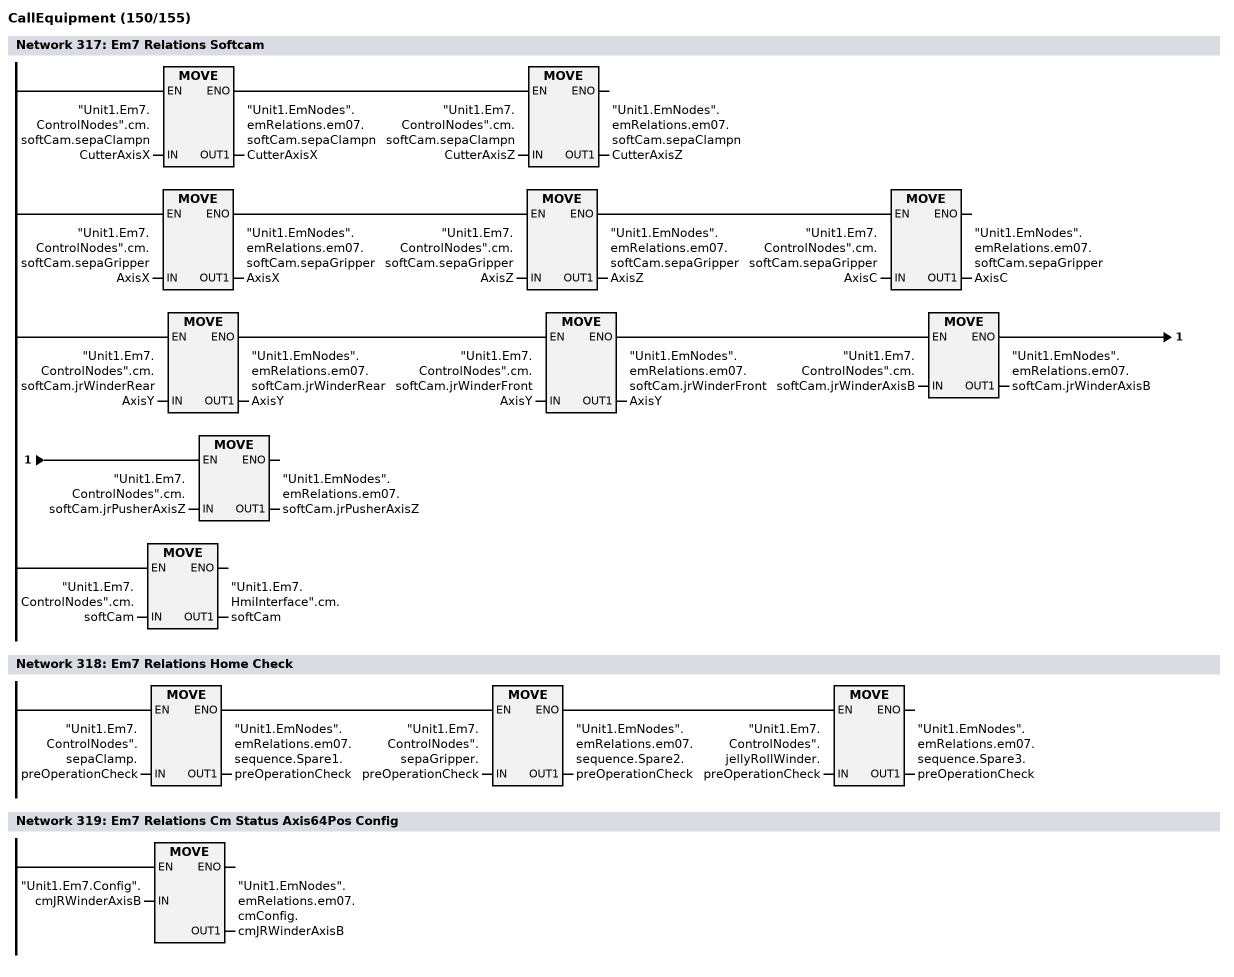
   RUNG wire#powerrail
      Move(in := "Unit1.Em7.ControlNodes".cm.softCam.sepaClampnCutterAxisX, out1 => "Unit1.EmNodes".emRelations.em07.softCam.sepaClampnCutterAxisX)
      Move(in := "Unit1.Em7.ControlNodes".cm.softCam.sepaClampnCutterAxisZ, out1 => "Unit1.EmNodes".emRelations.em07.softCam.sepaClampnCutterAxisZ)
   END_RUNG
   RUNG wire#powerrail
      Move(in := "Unit1.Em7.ControlNodes".cm.softCam.sepaGripperAxisX, out1 => "Unit1.EmNodes".emRelations.em07.softCam.sepaGripperAxisX)
      Move(in := "Unit1.Em7.ControlNodes".cm.softCam.sepaGripperAxisZ, out1 => "Unit1.EmNodes".emRelations.em07.softCam.sepaGripperAxisZ)
      Move(in := "Unit1.Em7.ControlNodes".cm.softCam.sepaGripperAxisC, out1 => "Unit1.EmNodes".emRelations.em07.softCam.sepaGripperAxisC)
   END_RUNG
   RUNG wire#powerrail
      Move(in := "Unit1.Em7.ControlNodes".cm.softCam.jrWinderRearAxisY, out1 => "Unit1.EmNodes".emRelations.em07.softCam.jrWinderRearAxisY)
      Move(in := "Unit1.Em7.ControlNodes".cm.softCam.jrWinderFrontAxisY, out1 => "Unit1.EmNodes".emRelations.em07.softCam.jrWinderFrontAxisY)
      Move(in := "Unit1.Em7.ControlNodes".cm.softCam.jrWinderAxisB, out1 => "Unit1.EmNodes".emRelations.em07.softCam.jrWinderAxisB)
      Move(in := "Unit1.Em7.ControlNodes".cm.softCam.jrPusherAxisZ, out1 => "Unit1.EmNodes".emRelations.em07.softCam.jrPusherAxisZ)
   END_RUNG
   RUNG wire#powerrail
      Move(in := "Unit1.Em7.ControlNodes".cm.softCam, out1 => "Unit1.Em7.HmiInterface".cm.softCam)
   END_RUNG
   // the same network as SCL:
   "Unit1.EmNodes".emRelations.em07.softCam.sepaClampnCutterAxisX := "Unit1.Em7.ControlNodes".cm.softCam.sepaClampnCutterAxisX;
   "Unit1.EmNodes".emRelations.em07.softCam.sepaClampnCutterAxisZ := "Unit1.Em7.ControlNodes".cm.softCam.sepaClampnCutterAxisZ;
   "Unit1.EmNodes".emRelations.em07.softCam.sepaGripperAxisX := "Unit1.Em7.ControlNodes".cm.softCam.sepaGripperAxisX;
   "Unit1.EmNodes".emRelations.em07.softCam.sepaGripperAxisZ := "Unit1.Em7.ControlNodes".cm.softCam.sepaGripperAxisZ;
   "Unit1.EmNodes".emRelations.em07.softCam.sepaGripperAxisC := "Unit1.Em7.ControlNodes".cm.softCam.sepaGripperAxisC;
   "Unit1.EmNodes".emRelations.em07.softCam.jrWinderRearAxisY := "Unit1.Em7.ControlNodes".cm.softCam.jrWinderRearAxisY;
   "Unit1.EmNodes".emRelations.em07.softCam.jrWinderFrontAxisY := "Unit1.Em7.ControlNodes".cm.softCam.jrWinderFrontAxisY;
   "Unit1.EmNodes".emRelations.em07.softCam.jrWinderAxisB := "Unit1.Em7.ControlNodes".cm.softCam.jrWinderAxisB;
   "Unit1.EmNodes".emRelations.em07.softCam.jrPusherAxisZ := "Unit1.Em7.ControlNodes".cm.softCam.jrPusherAxisZ;
   "Unit1.Em7.HmiInterface".cm.softCam := "Unit1.Em7.ControlNodes".cm.softCam;
END_REGION

REGION Network 318: Em7 Relations Home Check
   RUNG wire#powerrail
      Move(in := "Unit1.Em7.ControlNodes".sepaClamp.preOperationCheck, out1 => "Unit1.EmNodes".emRelations.em07.sequence.Spare1.preOperationCheck)
      Move(in := "Unit1.Em7.ControlNodes".sepaGripper.preOperationCheck, out1 => "Unit1.EmNodes".emRelations.em07.sequence.Spare2.preOperationCheck)
      Move(in := "Unit1.Em7.ControlNodes".jellyRollWinder.preOperationCheck, out1 => "Unit1.EmNodes".emRelations.em07.sequence.Spare3.preOperationCheck)
   END_RUNG
   // the same network as SCL:
   "Unit1.EmNodes".emRelations.em07.sequence.Spare1.preOperationCheck := "Unit1.Em7.ControlNodes".sepaClamp.preOperationCheck;
   "Unit1.EmNodes".emRelations.em07.sequence.Spare2.preOperationCheck := "Unit1.Em7.ControlNodes".sepaGripper.preOperationCheck;
   "Unit1.EmNodes".emRelations.em07.sequence.Spare3.preOperationCheck := "Unit1.Em7.ControlNodes".jellyRollWinder.preOperationCheck;
END_REGION

REGION Network 319: Em7 Relations Cm Status Axis64Pos Config
   RUNG wire#powerrail
      Move(in := "Unit1.Em7.Config".cmJRWinderAxisB, out1 => "Unit1.EmNodes".emRelations.em07.cmConfig.cmJRWinderAxisB)
   END_RUNG
   // the same network as SCL:
   "Unit1.EmNodes".emRelations.em07.cmConfig.cmJRWinderAxisB := "Unit1.Em7.Config".cmJRWinderAxisB;
END_REGION

REGION Network 320: Em7 Relations Cm Status Cylinder
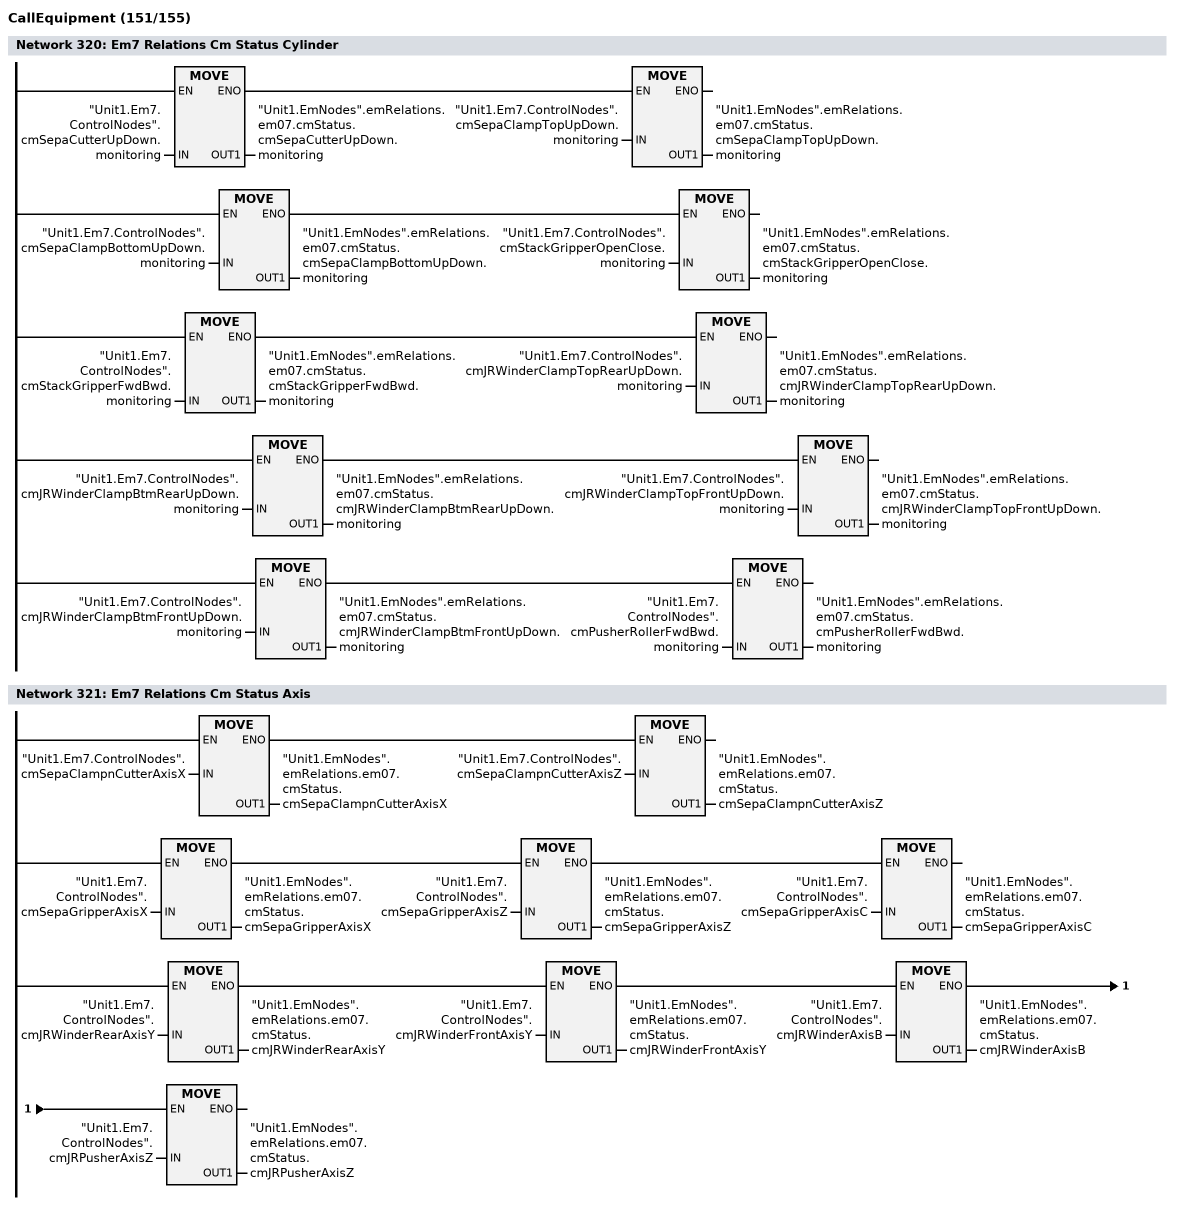
   RUNG wire#powerrail
      Move(in := "Unit1.Em7.ControlNodes".cmSepaCutterUpDown.monitoring, out1 => "Unit1.EmNodes".emRelations.em07.cmStatus.cmSepaCutterUpDown.monitoring)
      Move(in := "Unit1.Em7.ControlNodes".cmSepaClampTopUpDown.monitoring, out1 => "Unit1.EmNodes".emRelations.em07.cmStatus.cmSepaClampTopUpDown.monitoring)
   END_RUNG
   RUNG wire#powerrail
      Move(in := "Unit1.Em7.ControlNodes".cmSepaClampBottomUpDown.monitoring, out1 => "Unit1.EmNodes".emRelations.em07.cmStatus.cmSepaClampBottomUpDown.monitoring)
      Move(in := "Unit1.Em7.ControlNodes".cmStackGripperOpenClose.monitoring, out1 => "Unit1.EmNodes".emRelations.em07.cmStatus.cmStackGripperOpenClose.monitoring)
   END_RUNG
   RUNG wire#powerrail
      Move(in := "Unit1.Em7.ControlNodes".cmStackGripperFwdBwd.monitoring, out1 => "Unit1.EmNodes".emRelations.em07.cmStatus.cmStackGripperFwdBwd.monitoring)
      Move(in := "Unit1.Em7.ControlNodes".cmJRWinderClampTopRearUpDown.monitoring, out1 => "Unit1.EmNodes".emRelations.em07.cmStatus.cmJRWinderClampTopRearUpDown.monitoring)
   END_RUNG
   RUNG wire#powerrail
      Move(in := "Unit1.Em7.ControlNodes".cmJRWinderClampBtmRearUpDown.monitoring, out1 => "Unit1.EmNodes".emRelations.em07.cmStatus.cmJRWinderClampBtmRearUpDown.monitoring)
      Move(in := "Unit1.Em7.ControlNodes".cmJRWinderClampTopFrontUpDown.monitoring, out1 => "Unit1.EmNodes".emRelations.em07.cmStatus.cmJRWinderClampTopFrontUpDown.monitoring)
   END_RUNG
   RUNG wire#powerrail
      Move(in := "Unit1.Em7.ControlNodes".cmJRWinderClampBtmFrontUpDown.monitoring, out1 => "Unit1.EmNodes".emRelations.em07.cmStatus.cmJRWinderClampBtmFrontUpDown.monitoring)
      Move(in := "Unit1.Em7.ControlNodes".cmPusherRollerFwdBwd.monitoring, out1 => "Unit1.EmNodes".emRelations.em07.cmStatus.cmPusherRollerFwdBwd.monitoring)
   END_RUNG
   // the same network as SCL:
   "Unit1.EmNodes".emRelations.em07.cmStatus.cmSepaCutterUpDown.monitoring := "Unit1.Em7.ControlNodes".cmSepaCutterUpDown.monitoring;
   "Unit1.EmNodes".emRelations.em07.cmStatus.cmSepaClampTopUpDown.monitoring := "Unit1.Em7.ControlNodes".cmSepaClampTopUpDown.monitoring;
   "Unit1.EmNodes".emRelations.em07.cmStatus.cmSepaClampBottomUpDown.monitoring := "Unit1.Em7.ControlNodes".cmSepaClampBottomUpDown.monitoring;
   "Unit1.EmNodes".emRelations.em07.cmStatus.cmStackGripperOpenClose.monitoring := "Unit1.Em7.ControlNodes".cmStackGripperOpenClose.monitoring;
   "Unit1.EmNodes".emRelations.em07.cmStatus.cmStackGripperFwdBwd.monitoring := "Unit1.Em7.ControlNodes".cmStackGripperFwdBwd.monitoring;
   "Unit1.EmNodes".emRelations.em07.cmStatus.cmJRWinderClampTopRearUpDown.monitoring := "Unit1.Em7.ControlNodes".cmJRWinderClampTopRearUpDown.monitoring;
   "Unit1.EmNodes".emRelations.em07.cmStatus.cmJRWinderClampBtmRearUpDown.monitoring := "Unit1.Em7.ControlNodes".cmJRWinderClampBtmRearUpDown.monitoring;
   "Unit1.EmNodes".emRelations.em07.cmStatus.cmJRWinderClampTopFrontUpDown.monitoring := "Unit1.Em7.ControlNodes".cmJRWinderClampTopFrontUpDown.monitoring;
   "Unit1.EmNodes".emRelations.em07.cmStatus.cmJRWinderClampBtmFrontUpDown.monitoring := "Unit1.Em7.ControlNodes".cmJRWinderClampBtmFrontUpDown.monitoring;
   "Unit1.EmNodes".emRelations.em07.cmStatus.cmPusherRollerFwdBwd.monitoring := "Unit1.Em7.ControlNodes".cmPusherRollerFwdBwd.monitoring;
END_REGION

REGION Network 321: Em7 Relations Cm Status Axis
   RUNG wire#powerrail
      Move(in := "Unit1.Em7.ControlNodes".cmSepaClampnCutterAxisX, out1 => "Unit1.EmNodes".emRelations.em07.cmStatus.cmSepaClampnCutterAxisX)
      Move(in := "Unit1.Em7.ControlNodes".cmSepaClampnCutterAxisZ, out1 => "Unit1.EmNodes".emRelations.em07.cmStatus.cmSepaClampnCutterAxisZ)
   END_RUNG
   RUNG wire#powerrail
      Move(in := "Unit1.Em7.ControlNodes".cmSepaGripperAxisX, out1 => "Unit1.EmNodes".emRelations.em07.cmStatus.cmSepaGripperAxisX)
      Move(in := "Unit1.Em7.ControlNodes".cmSepaGripperAxisZ, out1 => "Unit1.EmNodes".emRelations.em07.cmStatus.cmSepaGripperAxisZ)
      Move(in := "Unit1.Em7.ControlNodes".cmSepaGripperAxisC, out1 => "Unit1.EmNodes".emRelations.em07.cmStatus.cmSepaGripperAxisC)
   END_RUNG
   RUNG wire#powerrail
      Move(in := "Unit1.Em7.ControlNodes".cmJRWinderRearAxisY, out1 => "Unit1.EmNodes".emRelations.em07.cmStatus.cmJRWinderRearAxisY)
      Move(in := "Unit1.Em7.ControlNodes".cmJRWinderFrontAxisY, out1 => "Unit1.EmNodes".emRelations.em07.cmStatus.cmJRWinderFrontAxisY)
      Move(in := "Unit1.Em7.ControlNodes".cmJRWinderAxisB, out1 => "Unit1.EmNodes".emRelations.em07.cmStatus.cmJRWinderAxisB)
      Move(in := "Unit1.Em7.ControlNodes".cmJRPusherAxisZ, out1 => "Unit1.EmNodes".emRelations.em07.cmStatus.cmJRPusherAxisZ)
   END_RUNG
   // the same network as SCL:
   "Unit1.EmNodes".emRelations.em07.cmStatus.cmSepaClampnCutterAxisX := "Unit1.Em7.ControlNodes".cmSepaClampnCutterAxisX;
   "Unit1.EmNodes".emRelations.em07.cmStatus.cmSepaClampnCutterAxisZ := "Unit1.Em7.ControlNodes".cmSepaClampnCutterAxisZ;
   "Unit1.EmNodes".emRelations.em07.cmStatus.cmSepaGripperAxisX := "Unit1.Em7.ControlNodes".cmSepaGripperAxisX;
   "Unit1.EmNodes".emRelations.em07.cmStatus.cmSepaGripperAxisZ := "Unit1.Em7.ControlNodes".cmSepaGripperAxisZ;
   "Unit1.EmNodes".emRelations.em07.cmStatus.cmSepaGripperAxisC := "Unit1.Em7.ControlNodes".cmSepaGripperAxisC;
   "Unit1.EmNodes".emRelations.em07.cmStatus.cmJRWinderRearAxisY := "Unit1.Em7.ControlNodes".cmJRWinderRearAxisY;
   "Unit1.EmNodes".emRelations.em07.cmStatus.cmJRWinderFrontAxisY := "Unit1.Em7.ControlNodes".cmJRWinderFrontAxisY;
   "Unit1.EmNodes".emRelations.em07.cmStatus.cmJRWinderAxisB := "Unit1.Em7.ControlNodes".cmJRWinderAxisB;
   "Unit1.EmNodes".emRelations.em07.cmStatus.cmJRPusherAxisZ := "Unit1.Em7.ControlNodes".cmJRPusherAxisZ;
END_REGION

REGION Network 322: Em7 Relations Cm Status Digital Signal
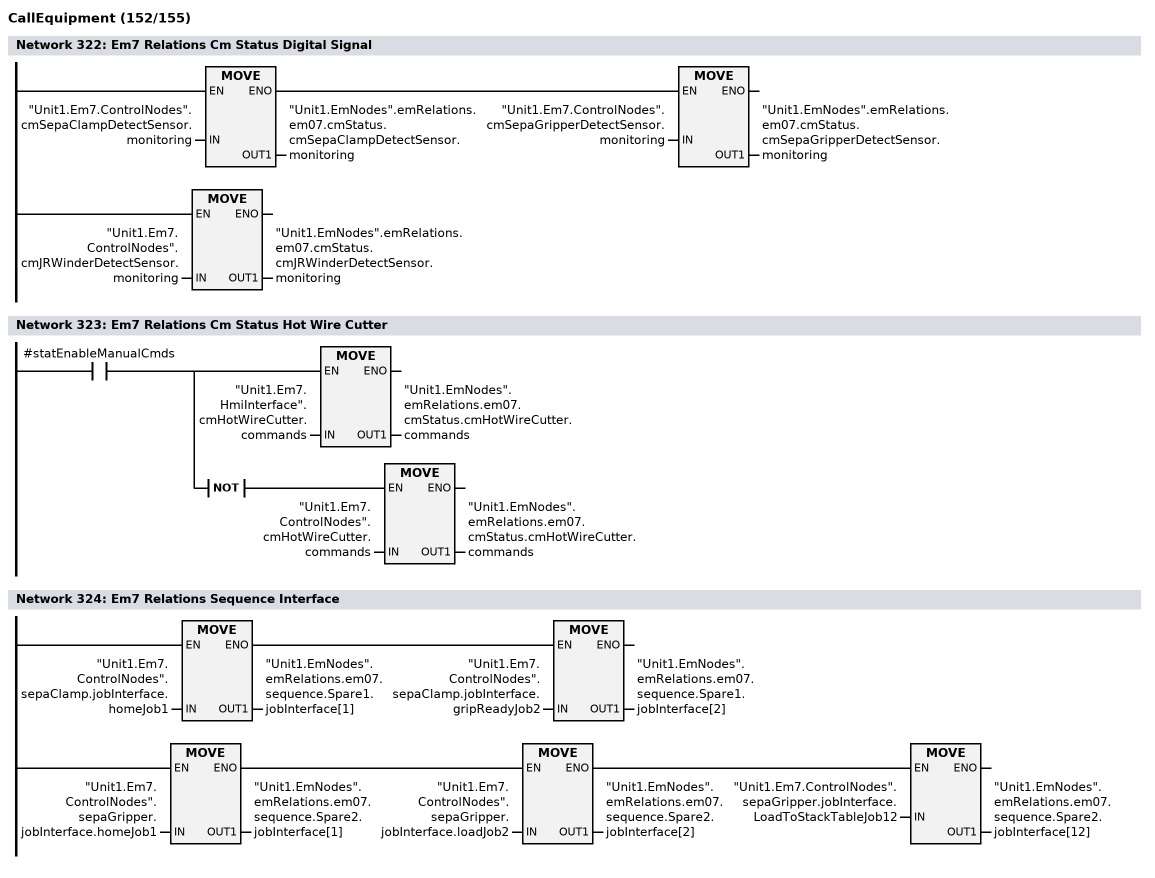
   RUNG wire#powerrail
      Move(in := "Unit1.Em7.ControlNodes".cmSepaClampDetectSensor.monitoring, out1 => "Unit1.EmNodes".emRelations.em07.cmStatus.cmSepaClampDetectSensor.monitoring)
      Move(in := "Unit1.Em7.ControlNodes".cmSepaGripperDetectSensor.monitoring, out1 => "Unit1.EmNodes".emRelations.em07.cmStatus.cmSepaGripperDetectSensor.monitoring)
   END_RUNG
   RUNG wire#powerrail
      Move(in := "Unit1.Em7.ControlNodes".cmJRWinderDetectSensor.monitoring, out1 => "Unit1.EmNodes".emRelations.em07.cmStatus.cmJRWinderDetectSensor.monitoring)
   END_RUNG
   // the same network as SCL:
   "Unit1.EmNodes".emRelations.em07.cmStatus.cmSepaClampDetectSensor.monitoring := "Unit1.Em7.ControlNodes".cmSepaClampDetectSensor.monitoring;
   "Unit1.EmNodes".emRelations.em07.cmStatus.cmSepaGripperDetectSensor.monitoring := "Unit1.Em7.ControlNodes".cmSepaGripperDetectSensor.monitoring;
   "Unit1.EmNodes".emRelations.em07.cmStatus.cmJRWinderDetectSensor.monitoring := "Unit1.Em7.ControlNodes".cmJRWinderDetectSensor.monitoring;
END_REGION

REGION Network 323: Em7 Relations Cm Status Hot Wire Cutter
   RUNG wire#powerrail
      Contact( #statEnableManualCmds )
      wire#w1
      Move(in := "Unit1.Em7.HmiInterface".cmHotWireCutter.commands, out1 => "Unit1.EmNodes".emRelations.em07.cmStatus.cmHotWireCutter.commands)
   END_RUNG
   RUNG wire#w1
      Not()
      Move(in := "Unit1.Em7.ControlNodes".cmHotWireCutter.commands, out1 => "Unit1.EmNodes".emRelations.em07.cmStatus.cmHotWireCutter.commands)
   END_RUNG
   // the same network as SCL:
   IF #statEnableManualCmds THEN
       "Unit1.EmNodes".emRelations.em07.cmStatus.cmHotWireCutter.commands := "Unit1.Em7.HmiInterface".cmHotWireCutter.commands;
   END_IF;
   IF NOT #statEnableManualCmds THEN
       "Unit1.EmNodes".emRelations.em07.cmStatus.cmHotWireCutter.commands := "Unit1.Em7.ControlNodes".cmHotWireCutter.commands;
   END_IF;
END_REGION

REGION Network 324: Em7 Relations Sequence Interface
   RUNG wire#powerrail
      Move(in := "Unit1.Em7.ControlNodes".sepaClamp.jobInterface.homeJob1, out1 => "Unit1.EmNodes".emRelations.em07.sequence.Spare1.jobInterface[1])
      Move(in := "Unit1.Em7.ControlNodes".sepaClamp.jobInterface.gripReadyJob2, out1 => "Unit1.EmNodes".emRelations.em07.sequence.Spare1.jobInterface[2])
   END_RUNG
   RUNG wire#powerrail
      Move(in := "Unit1.Em7.ControlNodes".sepaGripper.jobInterface.homeJob1, out1 => "Unit1.EmNodes".emRelations.em07.sequence.Spare2.jobInterface[1])
      Move(in := "Unit1.Em7.ControlNodes".sepaGripper.jobInterface.loadJob2, out1 => "Unit1.EmNodes".emRelations.em07.sequence.Spare2.jobInterface[2])
      Move(in := "Unit1.Em7.ControlNodes".sepaGripper.jobInterface.LoadToStackTableJob12, out1 => "Unit1.EmNodes".emRelations.em07.sequence.Spare2.jobInterface[12])
   END_RUNG
   // the same network as SCL:
   "Unit1.EmNodes".emRelations.em07.sequence.Spare1.jobInterface[1] := "Unit1.Em7.ControlNodes".sepaClamp.jobInterface.homeJob1;
   "Unit1.EmNodes".emRelations.em07.sequence.Spare1.jobInterface[2] := "Unit1.Em7.ControlNodes".sepaClamp.jobInterface.gripReadyJob2;
   "Unit1.EmNodes".emRelations.em07.sequence.Spare2.jobInterface[1] := "Unit1.Em7.ControlNodes".sepaGripper.jobInterface.homeJob1;
   "Unit1.EmNodes".emRelations.em07.sequence.Spare2.jobInterface[2] := "Unit1.Em7.ControlNodes".sepaGripper.jobInterface.loadJob2;
   "Unit1.EmNodes".emRelations.em07.sequence.Spare2.jobInterface[12] := "Unit1.Em7.ControlNodes".sepaGripper.jobInterface.LoadToStackTableJob12;
END_REGION

REGION Network 325: Em Nodes Brake Test
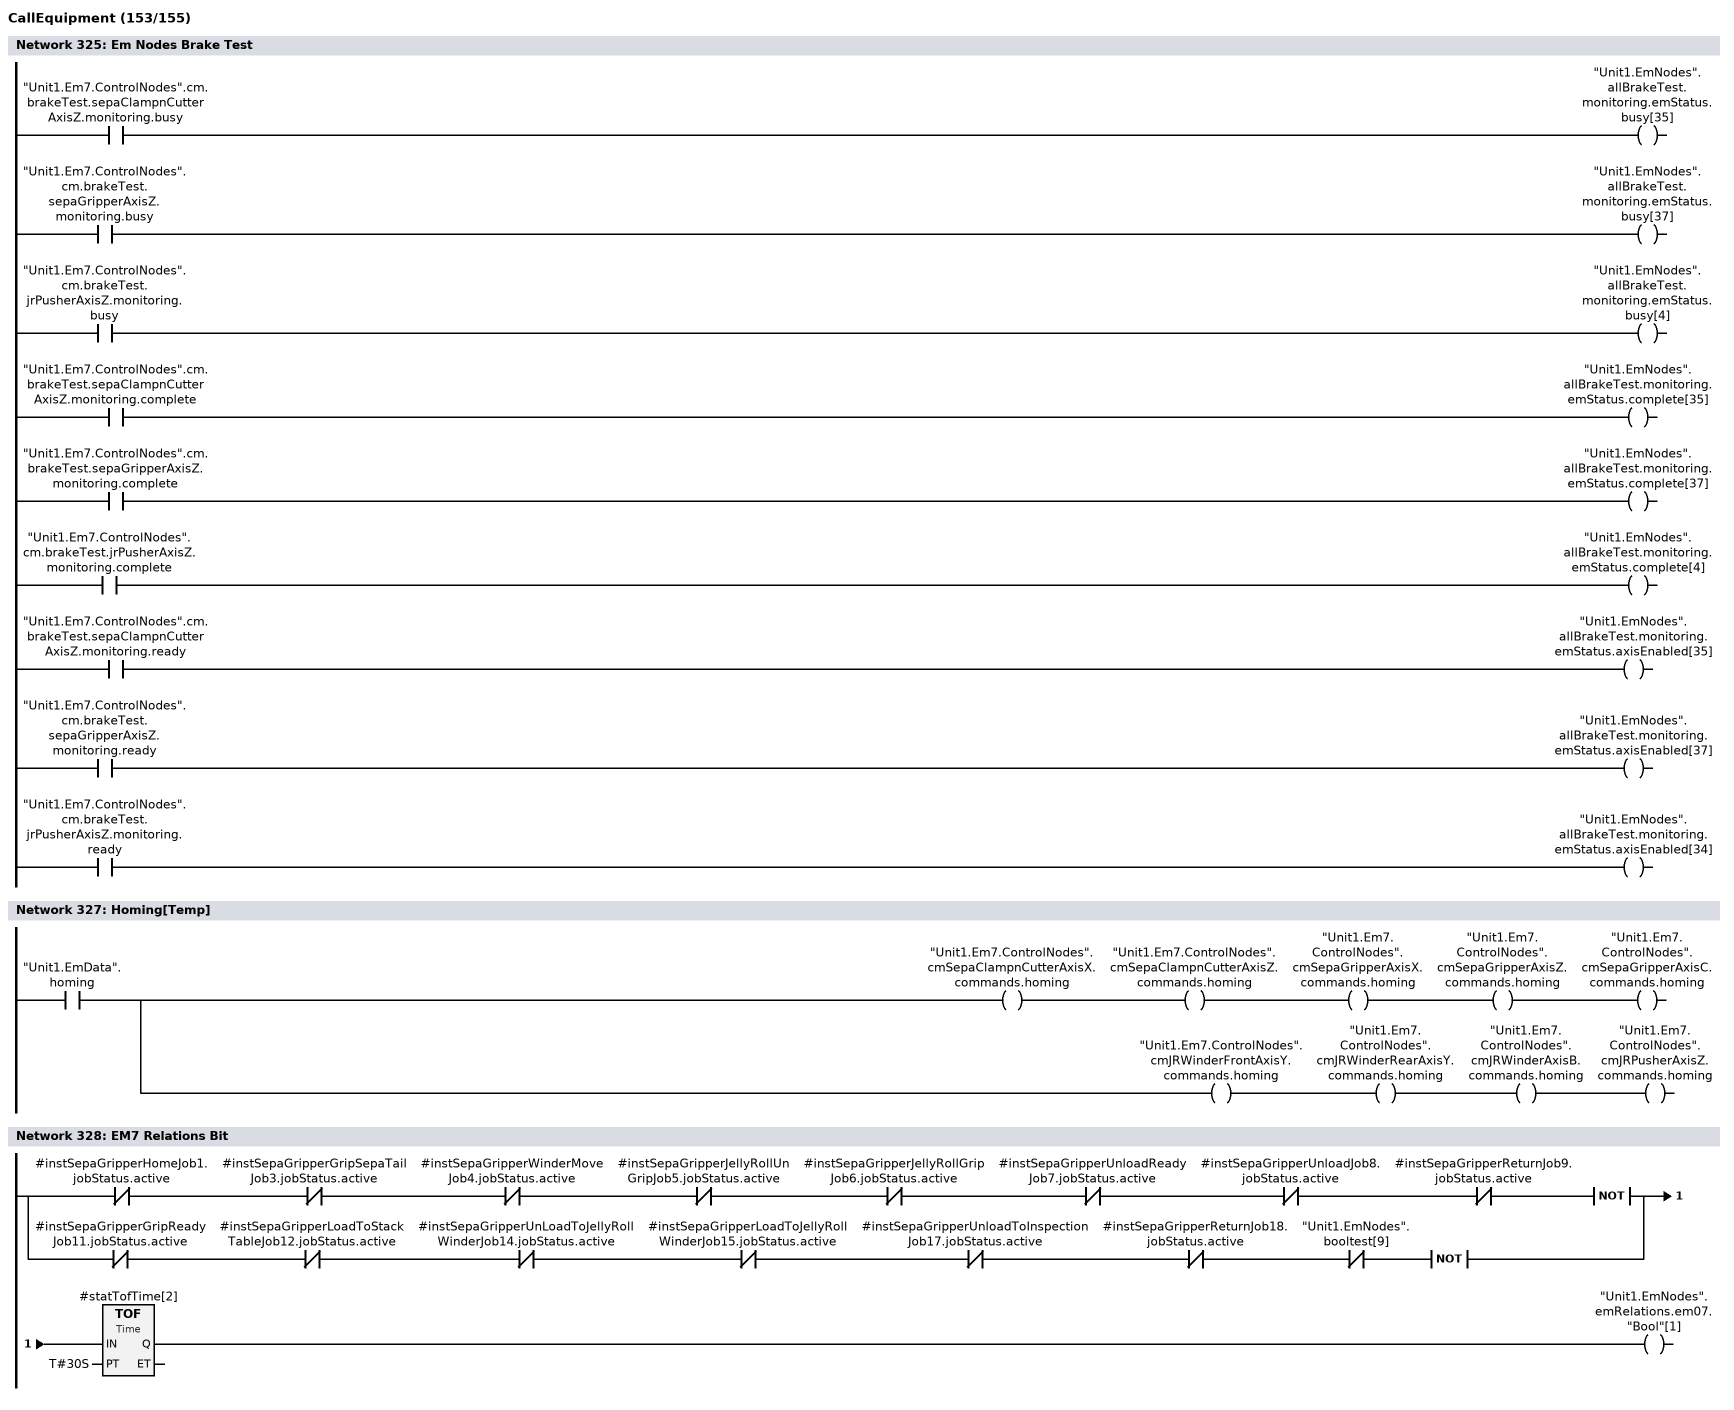
   RUNG wire#powerrail
      Contact( "Unit1.Em7.ControlNodes".cm.brakeTest.sepaClampnCutterAxisZ.monitoring.busy )
      Coil( "Unit1.EmNodes".allBrakeTest.monitoring.emStatus.busy[35] )
   END_RUNG
   RUNG wire#powerrail
      Contact( "Unit1.Em7.ControlNodes".cm.brakeTest.sepaGripperAxisZ.monitoring.busy )
      Coil( "Unit1.EmNodes".allBrakeTest.monitoring.emStatus.busy[37] )
   END_RUNG
   RUNG wire#powerrail
      Contact( "Unit1.Em7.ControlNodes".cm.brakeTest.jrPusherAxisZ.monitoring.busy )
      Coil( "Unit1.EmNodes".allBrakeTest.monitoring.emStatus.busy[4] )
   END_RUNG
   RUNG wire#powerrail
      Contact( "Unit1.Em7.ControlNodes".cm.brakeTest.sepaClampnCutterAxisZ.monitoring.complete )
      Coil( "Unit1.EmNodes".allBrakeTest.monitoring.emStatus.complete[35] )
   END_RUNG
   RUNG wire#powerrail
      Contact( "Unit1.Em7.ControlNodes".cm.brakeTest.sepaGripperAxisZ.monitoring.complete )
      Coil( "Unit1.EmNodes".allBrakeTest.monitoring.emStatus.complete[37] )
   END_RUNG
   RUNG wire#powerrail
      Contact( "Unit1.Em7.ControlNodes".cm.brakeTest.jrPusherAxisZ.monitoring.complete )
      Coil( "Unit1.EmNodes".allBrakeTest.monitoring.emStatus.complete[4] )
   END_RUNG
   RUNG wire#powerrail
      Contact( "Unit1.Em7.ControlNodes".cm.brakeTest.sepaClampnCutterAxisZ.monitoring.ready )
      Coil( "Unit1.EmNodes".allBrakeTest.monitoring.emStatus.axisEnabled[35] )
   END_RUNG
   RUNG wire#powerrail
      Contact( "Unit1.Em7.ControlNodes".cm.brakeTest.sepaGripperAxisZ.monitoring.ready )
      Coil( "Unit1.EmNodes".allBrakeTest.monitoring.emStatus.axisEnabled[37] )
   END_RUNG
   RUNG wire#powerrail
      Contact( "Unit1.Em7.ControlNodes".cm.brakeTest.jrPusherAxisZ.monitoring.ready )
      Coil( "Unit1.EmNodes".allBrakeTest.monitoring.emStatus.axisEnabled[34] )
   END_RUNG
   // the same network as SCL:
   "Unit1.EmNodes".allBrakeTest.monitoring.emStatus.busy[35] := "Unit1.Em7.ControlNodes".cm.brakeTest.sepaClampnCutterAxisZ.monitoring.busy;
   "Unit1.EmNodes".allBrakeTest.monitoring.emStatus.busy[37] := "Unit1.Em7.ControlNodes".cm.brakeTest.sepaGripperAxisZ.monitoring.busy;
   "Unit1.EmNodes".allBrakeTest.monitoring.emStatus.busy[4] := "Unit1.Em7.ControlNodes".cm.brakeTest.jrPusherAxisZ.monitoring.busy;
   "Unit1.EmNodes".allBrakeTest.monitoring.emStatus.complete[35] := "Unit1.Em7.ControlNodes".cm.brakeTest.sepaClampnCutterAxisZ.monitoring.complete;
   "Unit1.EmNodes".allBrakeTest.monitoring.emStatus.complete[37] := "Unit1.Em7.ControlNodes".cm.brakeTest.sepaGripperAxisZ.monitoring.complete;
   "Unit1.EmNodes".allBrakeTest.monitoring.emStatus.complete[4] := "Unit1.Em7.ControlNodes".cm.brakeTest.jrPusherAxisZ.monitoring.complete;
   "Unit1.EmNodes".allBrakeTest.monitoring.emStatus.axisEnabled[35] := "Unit1.Em7.ControlNodes".cm.brakeTest.sepaClampnCutterAxisZ.monitoring.ready;
   "Unit1.EmNodes".allBrakeTest.monitoring.emStatus.axisEnabled[37] := "Unit1.Em7.ControlNodes".cm.brakeTest.sepaGripperAxisZ.monitoring.ready;
   "Unit1.EmNodes".allBrakeTest.monitoring.emStatus.axisEnabled[34] := "Unit1.Em7.ControlNodes".cm.brakeTest.jrPusherAxisZ.monitoring.ready;
END_REGION

REGION Network 326: Em Nodes BA060 Communication
END_REGION

REGION Network 327: Homing[Temp]
   RUNG wire#powerrail
      Contact( "Unit1.EmData".homing )
      wire#w1
      Coil( "Unit1.Em7.ControlNodes".cmSepaClampnCutterAxisX.commands.homing )
      Coil( "Unit1.Em7.ControlNodes".cmSepaClampnCutterAxisZ.commands.homing )
      Coil( "Unit1.Em7.ControlNodes".cmSepaGripperAxisX.commands.homing )
      Coil( "Unit1.Em7.ControlNodes".cmSepaGripperAxisZ.commands.homing )
      Coil( "Unit1.Em7.ControlNodes".cmSepaGripperAxisC.commands.homing )
   END_RUNG
   RUNG wire#w1
      Coil( "Unit1.Em7.ControlNodes".cmJRWinderFrontAxisY.commands.homing )
      Coil( "Unit1.Em7.ControlNodes".cmJRWinderRearAxisY.commands.homing )
      Coil( "Unit1.Em7.ControlNodes".cmJRWinderAxisB.commands.homing )
      Coil( "Unit1.Em7.ControlNodes".cmJRPusherAxisZ.commands.homing )
   END_RUNG
   // the same network as SCL:
   "Unit1.Em7.ControlNodes".cmSepaClampnCutterAxisX.commands.homing := "Unit1.EmData".homing;
   "Unit1.Em7.ControlNodes".cmSepaClampnCutterAxisZ.commands.homing := "Unit1.EmData".homing;
   "Unit1.Em7.ControlNodes".cmSepaGripperAxisX.commands.homing := "Unit1.EmData".homing;
   "Unit1.Em7.ControlNodes".cmSepaGripperAxisZ.commands.homing := "Unit1.EmData".homing;
   "Unit1.Em7.ControlNodes".cmSepaGripperAxisC.commands.homing := "Unit1.EmData".homing;
   "Unit1.Em7.ControlNodes".cmJRWinderFrontAxisY.commands.homing := "Unit1.EmData".homing;
   "Unit1.Em7.ControlNodes".cmJRWinderRearAxisY.commands.homing := "Unit1.EmData".homing;
   "Unit1.Em7.ControlNodes".cmJRWinderAxisB.commands.homing := "Unit1.EmData".homing;
   "Unit1.Em7.ControlNodes".cmJRPusherAxisZ.commands.homing := "Unit1.EmData".homing;
END_REGION

REGION Network 328: EM7 Relations Bit
   RUNG wire#powerrail
      I_Contact( #instSepaGripperHomeJob1.jobStatus.active )
      I_Contact( #instSepaGripperGripSepaTailJob3.jobStatus.active )
      I_Contact( #instSepaGripperWinderMoveJob4.jobStatus.active )
      I_Contact( #instSepaGripperJellyRollUnGripJob5.jobStatus.active )
      I_Contact( #instSepaGripperJellyRollGripJob6.jobStatus.active )
      I_Contact( #instSepaGripperUnloadReadyJob7.jobStatus.active )
      I_Contact( #instSepaGripperUnloadJob8.jobStatus.active )
      I_Contact( #instSepaGripperReturnJob9.jobStatus.active )
      Not()
      wire#w1
      { S7_Templates := "time_type := Time" } #statTofTime[2].TOF(pt := T#30S, et =>)
      Coil( "Unit1.EmNodes".emRelations.em07."Bool"[1] )
   END_RUNG
   RUNG wire#powerrail
      I_Contact( #instSepaGripperGripReadyJob11.jobStatus.active )
      I_Contact( #instSepaGripperLoadToStackTableJob12.jobStatus.active )
      I_Contact( #instSepaGripperUnLoadToJellyRollWinderJob14.jobStatus.active )
      I_Contact( #instSepaGripperLoadToJellyRollWinderJob15.jobStatus.active )
      I_Contact( #instSepaGripperUnloadToInspectionJob17.jobStatus.active )
      I_Contact( #instSepaGripperReturnJob18.jobStatus.active )
      I_Contact( "Unit1.EmNodes".booltest[9] )
      Not()
   END_RUNG wire#w1
   // the same network as SCL:
   #statTofTime[2].TOF(IN := NOT (NOT #instSepaGripperHomeJob1.jobStatus.active AND NOT #instSepaGripperGripSepaTailJob3.jobStatus.active AND NOT #instSepaGripperWinderMoveJob4.jobStatus.active AND NOT #instSepaGripperJellyRollUnGripJob5.jobStatus.active AND NOT #instSepaGripperJellyRollGripJob6.jobStatus.active AND NOT #instSepaGripperUnloadReadyJob7.jobStatus.active AND NOT #instSepaGripperUnloadJob8.jobStatus.active AND NOT #instSepaGripperReturnJob9.jobStatus.active) OR NOT (NOT #instSepaGripperGripReadyJob11.jobStatus.active AND NOT #instSepaGripperLoadToStackTableJob12.jobStatus.active AND NOT #instSepaGripperUnLoadToJellyRollWinderJob14.jobStatus.active AND NOT #instSepaGripperLoadToJellyRollWinderJob15.jobStatus.active AND NOT #instSepaGripperUnloadToInspectionJob17.jobStatus.active AND NOT #instSepaGripperReturnJob18.jobStatus.active AND NOT "Unit1.EmNodes".booltest[9]),
                       PT := T#30S);
   "Unit1.EmNodes".emRelations.em07."Bool"[1] := #statTofTime[2].Q;
END_REGION

REGION Network 329
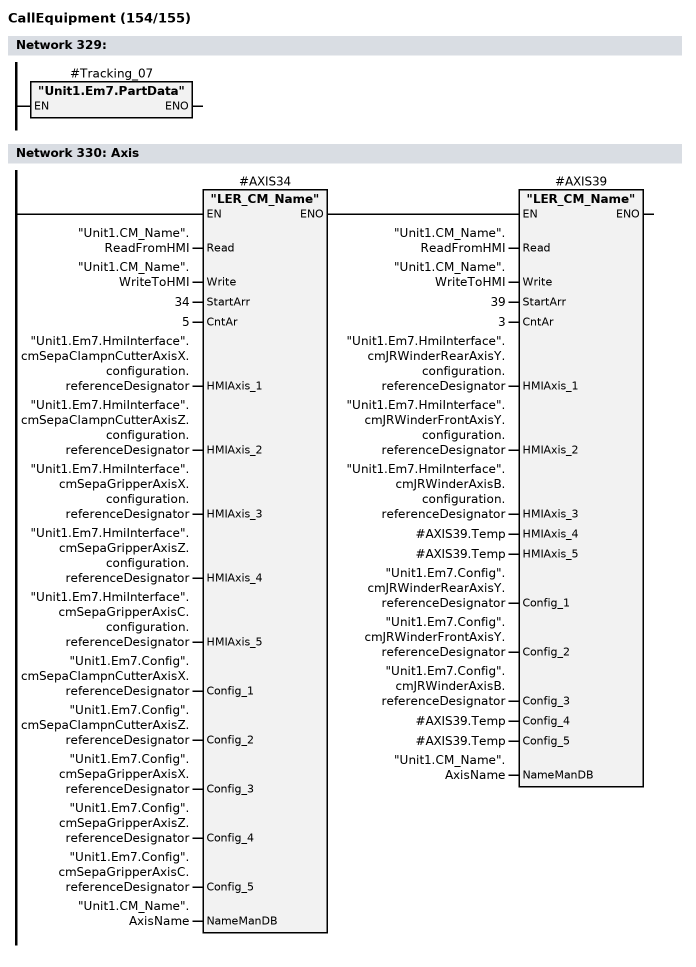
   RUNG wire#powerrail
      #Tracking_07()
   END_RUNG
   // the same network as SCL:
   #Tracking_07();   // "Unit1.Em7.PartData"
END_REGION

REGION Network 330: Axis
   RUNG wire#powerrail
      #AXIS34(Read := "Unit1.CM_Name".ReadFromHMI, Write := "Unit1.CM_Name".WriteToHMI, StartArr := 34, CntAr := 5, HMIAxis_1 := "Unit1.Em7.HmiInterface".cmSepaClampnCutterAxisX.configuration.referenceDesignator, HMIAxis_2 := "Unit1.Em7.HmiInterface".cmSepaClampnCutterAxisZ.configuration.referenceDesignator, HMIAxis_3 := "Unit1.Em7.HmiInterface".cmSepaGripperAxisX.configuration.referenceDesignator, HMIAxis_4 := "Unit1.Em7.HmiInterface".cmSepaGripperAxisZ.configuration.referenceDesignator, HMIAxis_5 := "Unit1.Em7.HmiInterface".cmSepaGripperAxisC.configuration.referenceDesignator, Config_1 := "Unit1.Em7.Config".cmSepaClampnCutterAxisX.referenceDesignator, Config_2 := "Unit1.Em7.Config".cmSepaClampnCutterAxisZ.referenceDesignator, Config_3 := "Unit1.Em7.Config".cmSepaGripperAxisX.referenceDesignator, Config_4 := "Unit1.Em7.Config".cmSepaGripperAxisZ.referenceDesignator, Config_5 := "Unit1.Em7.Config".cmSepaGripperAxisC.referenceDesignator, NameManDB := "Unit1.CM_Name".AxisName)
      #AXIS39(Read := "Unit1.CM_Name".ReadFromHMI, Write := "Unit1.CM_Name".WriteToHMI, StartArr := 39, CntAr := 3, HMIAxis_1 := "Unit1.Em7.HmiInterface".cmJRWinderRearAxisY.configuration.referenceDesignator, HMIAxis_2 := "Unit1.Em7.HmiInterface".cmJRWinderFrontAxisY.configuration.referenceDesignator, HMIAxis_3 := "Unit1.Em7.HmiInterface".cmJRWinderAxisB.configuration.referenceDesignator, HMIAxis_4 := #AXIS39.Temp, HMIAxis_5 := #AXIS39.Temp, Config_1 := "Unit1.Em7.Config".cmJRWinderRearAxisY.referenceDesignator, Config_2 := "Unit1.Em7.Config".cmJRWinderFrontAxisY.referenceDesignator, Config_3 := "Unit1.Em7.Config".cmJRWinderAxisB.referenceDesignator, Config_4 := #AXIS39.Temp, Config_5 := #AXIS39.Temp, NameManDB := "Unit1.CM_Name".AxisName)
   END_RUNG
   // the same network as SCL:
   #AXIS34(Read := "Unit1.CM_Name".ReadFromHMI,   // "LER_CM_Name"
           Write := "Unit1.CM_Name".WriteToHMI,
           StartArr := 34,
           CntAr := 5,
           HMIAxis_1 := "Unit1.Em7.HmiInterface".cmSepaClampnCutterAxisX.configuration.referenceDesignator,
           HMIAxis_2 := "Unit1.Em7.HmiInterface".cmSepaClampnCutterAxisZ.configuration.referenceDesignator,
           HMIAxis_3 := "Unit1.Em7.HmiInterface".cmSepaGripperAxisX.configuration.referenceDesignator,
           HMIAxis_4 := "Unit1.Em7.HmiInterface".cmSepaGripperAxisZ.configuration.referenceDesignator,
           HMIAxis_5 := "Unit1.Em7.HmiInterface".cmSepaGripperAxisC.configuration.referenceDesignator,
           Config_1 := "Unit1.Em7.Config".cmSepaClampnCutterAxisX.referenceDesignator,
           Config_2 := "Unit1.Em7.Config".cmSepaClampnCutterAxisZ.referenceDesignator,
           Config_3 := "Unit1.Em7.Config".cmSepaGripperAxisX.referenceDesignator,
           Config_4 := "Unit1.Em7.Config".cmSepaGripperAxisZ.referenceDesignator,
           Config_5 := "Unit1.Em7.Config".cmSepaGripperAxisC.referenceDesignator,
           NameManDB := "Unit1.CM_Name".AxisName,
           ENO => #_w1);
   IF #_w1 THEN
       #AXIS39(Read := "Unit1.CM_Name".ReadFromHMI,   // "LER_CM_Name"
               Write := "Unit1.CM_Name".WriteToHMI,
               StartArr := 39,
               CntAr := 3,
               HMIAxis_1 := "Unit1.Em7.HmiInterface".cmJRWinderRearAxisY.configuration.referenceDesignator,
               HMIAxis_2 := "Unit1.Em7.HmiInterface".cmJRWinderFrontAxisY.configuration.referenceDesignator,
               HMIAxis_3 := "Unit1.Em7.HmiInterface".cmJRWinderAxisB.configuration.referenceDesignator,
               HMIAxis_4 := #AXIS39.Temp,
               HMIAxis_5 := #AXIS39.Temp,
               Config_1 := "Unit1.Em7.Config".cmJRWinderRearAxisY.referenceDesignator,
               Config_2 := "Unit1.Em7.Config".cmJRWinderFrontAxisY.referenceDesignator,
               Config_3 := "Unit1.Em7.Config".cmJRWinderAxisB.referenceDesignator,
               Config_4 := #AXIS39.Temp,
               Config_5 := #AXIS39.Temp,
               NameManDB := "Unit1.CM_Name".AxisName);
   END_IF;
END_REGION

REGION Network 331: Cylinder
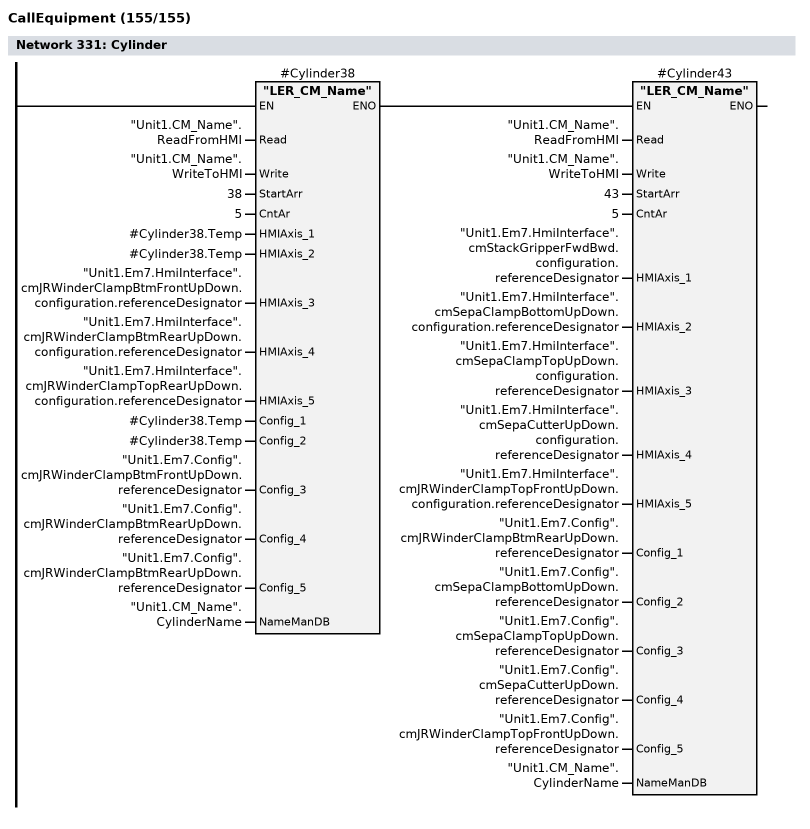
   RUNG wire#powerrail
      #Cylinder38(Read := "Unit1.CM_Name".ReadFromHMI, Write := "Unit1.CM_Name".WriteToHMI, StartArr := 38, CntAr := 5, HMIAxis_1 := #Cylinder38.Temp, HMIAxis_2 := #Cylinder38.Temp, HMIAxis_3 := "Unit1.Em7.HmiInterface".cmJRWinderClampBtmFrontUpDown.configuration.referenceDesignator, HMIAxis_4 := "Unit1.Em7.HmiInterface".cmJRWinderClampBtmRearUpDown.configuration.referenceDesignator, HMIAxis_5 := "Unit1.Em7.HmiInterface".cmJRWinderClampTopRearUpDown.configuration.referenceDesignator, Config_1 := #Cylinder38.Temp, Config_2 := #Cylinder38.Temp, Config_3 := "Unit1.Em7.Config".cmJRWinderClampBtmFrontUpDown.referenceDesignator, Config_4 := "Unit1.Em7.Config".cmJRWinderClampBtmRearUpDown.referenceDesignator, Config_5 := "Unit1.Em7.Config".cmJRWinderClampBtmRearUpDown.referenceDesignator, NameManDB := "Unit1.CM_Name".CylinderName)
      #Cylinder43(Read := "Unit1.CM_Name".ReadFromHMI, Write := "Unit1.CM_Name".WriteToHMI, StartArr := 43, CntAr := 5, HMIAxis_1 := "Unit1.Em7.HmiInterface".cmStackGripperFwdBwd.configuration.referenceDesignator, HMIAxis_2 := "Unit1.Em7.HmiInterface".cmSepaClampBottomUpDown.configuration.referenceDesignator, HMIAxis_3 := "Unit1.Em7.HmiInterface".cmSepaClampTopUpDown.configuration.referenceDesignator, HMIAxis_4 := "Unit1.Em7.HmiInterface".cmSepaCutterUpDown.configuration.referenceDesignator, HMIAxis_5 := "Unit1.Em7.HmiInterface".cmJRWinderClampTopFrontUpDown.configuration.referenceDesignator, Config_1 := "Unit1.Em7.Config".cmJRWinderClampBtmRearUpDown.referenceDesignator, Config_2 := "Unit1.Em7.Config".cmSepaClampBottomUpDown.referenceDesignator, Config_3 := "Unit1.Em7.Config".cmSepaClampTopUpDown.referenceDesignator, Config_4 := "Unit1.Em7.Config".cmSepaCutterUpDown.referenceDesignator, Config_5 := "Unit1.Em7.Config".cmJRWinderClampTopFrontUpDown.referenceDesignator, NameManDB := "Unit1.CM_Name".CylinderName)
   END_RUNG
   // the same network as SCL:
   #Cylinder38(Read := "Unit1.CM_Name".ReadFromHMI,   // "LER_CM_Name"
               Write := "Unit1.CM_Name".WriteToHMI,
               StartArr := 38,
               CntAr := 5,
               HMIAxis_1 := #Cylinder38.Temp,
               HMIAxis_2 := #Cylinder38.Temp,
               HMIAxis_3 := "Unit1.Em7.HmiInterface".cmJRWinderClampBtmFrontUpDown.configuration.referenceDesignator,
               HMIAxis_4 := "Unit1.Em7.HmiInterface".cmJRWinderClampBtmRearUpDown.configuration.referenceDesignator,
               HMIAxis_5 := "Unit1.Em7.HmiInterface".cmJRWinderClampTopRearUpDown.configuration.referenceDesignator,
               Config_1 := #Cylinder38.Temp,
               Config_2 := #Cylinder38.Temp,
               Config_3 := "Unit1.Em7.Config".cmJRWinderClampBtmFrontUpDown.referenceDesignator,
               Config_4 := "Unit1.Em7.Config".cmJRWinderClampBtmRearUpDown.referenceDesignator,
               Config_5 := "Unit1.Em7.Config".cmJRWinderClampBtmRearUpDown.referenceDesignator,
               NameManDB := "Unit1.CM_Name".CylinderName,
               ENO => #_w1);
   IF #_w1 THEN
       #Cylinder43(Read := "Unit1.CM_Name".ReadFromHMI,   // "LER_CM_Name"
                   Write := "Unit1.CM_Name".WriteToHMI,
                   StartArr := 43,
                   CntAr := 5,
                   HMIAxis_1 := "Unit1.Em7.HmiInterface".cmStackGripperFwdBwd.configuration.referenceDesignator,
                   HMIAxis_2 := "Unit1.Em7.HmiInterface".cmSepaClampBottomUpDown.configuration.referenceDesignator,
                   HMIAxis_3 := "Unit1.Em7.HmiInterface".cmSepaClampTopUpDown.configuration.referenceDesignator,
                   HMIAxis_4 := "Unit1.Em7.HmiInterface".cmSepaCutterUpDown.configuration.referenceDesignator,
                   HMIAxis_5 := "Unit1.Em7.HmiInterface".cmJRWinderClampTopFrontUpDown.configuration.referenceDesignator,
                   Config_1 := "Unit1.Em7.Config".cmJRWinderClampBtmRearUpDown.referenceDesignator,
                   Config_2 := "Unit1.Em7.Config".cmSepaClampBottomUpDown.referenceDesignator,
                   Config_3 := "Unit1.Em7.Config".cmSepaClampTopUpDown.referenceDesignator,
                   Config_4 := "Unit1.Em7.Config".cmSepaCutterUpDown.referenceDesignator,
                   Config_5 := "Unit1.Em7.Config".cmJRWinderClampTopFrontUpDown.referenceDesignator,
                   NameManDB := "Unit1.CM_Name".CylinderName);
   END_IF;
END_REGION
END_FUNCTION_BLOCK
